// TIA Portal project "Poao_V21" (V21)

(* hardware
DEVICE "S7-1200 station_1"  S7-1200 Station
   slot 0: "Rack_0"  S7-1200 Rack  Rack  V1.0
   slot 1: "PLC_2"  CPU 1214C DC/DC/DC  6ES7 214-1AG40-0XB0  V4.4
DEVICE "PC station"  SIMATIC PC station
   slot 0: "PC station"  Rail  SIMATIC PC-Station  V1.0
      slot 125: "Stationmanager"  Station_Manager  V6.0.4
   slot 1: "IE general_1"  IE General  IE_CP  V8.2.0
      slot 1: "PROFINET interface"  IEGeneral.Interface.8.2.0
   slot 3: "HMI_RT_1"  WinCC RT Advanced  6AV2 104-0xxxx-xxxx  17.0.0.0
      slot 33792: "主机接口"  Host interface
*)

// ===== PLC "PLC_2"  CPU 1214C DC/DC/DC =====

VAR_GLOBAL   // PLC tag table "默认变量表"
   "1层外呼上行指示灯" AT %M24.0 : Bool;
   "2层外呼上行指示灯" AT %M24.1 : Bool;
   "3层外呼上行指示灯" AT %M24.2 : Bool;
   "4层外呼上行指示灯" AT %M24.3 : Bool;
   "5层外呼上行指示灯" AT %M24.4 : Bool;
   "2层外呼下行指示灯" AT %M24.5 : Bool;
   "3层外呼下行指示灯" AT %M24.6 : Bool;
   "4层外呼下行指示灯" AT %M24.7 : Bool;
   "6层外呼下行指示灯" AT %M25.1 : Bool;
   "1号梯1层内呼指示灯" AT %M25.2 : Bool;
   "1号梯2层内呼指示灯" AT %M25.3 : Bool;
   "1号梯3层内呼指示灯" AT %M25.4 : Bool;
   "1号梯4层内呼指示灯" AT %M25.5 : Bool;
   "1号梯5层内呼指示灯" AT %M25.6 : Bool;
   "1号梯6层内呼指示灯" AT %M25.7 : Bool;
   "1号梯七段数码管a" AT %M26.2 : Bool;
   "1号梯七段数码管b" AT %M26.3 : Bool;
   "1号梯七段数码管c" AT %M26.4 : Bool;
   "1号梯七段数码管d" AT %M26.5 : Bool;
   "1号梯七段数码管e" AT %M26.6 : Bool;
   "1号梯七段数码管f" AT %M26.7 : Bool;
   "1号梯七段数码管g" AT %M33.7 : Bool;
   "1号梯上行指示" AT %M23.4 : Bool;
   "1号梯下行指示" AT %M2.5 : Bool;
   "1号梯电机启动信号" AT %M2.6 : Bool;
   "1号梯故障指示" AT %M23.5 : Bool;
   "1号梯照明指示" AT %M23.6 : Bool;
   "1号梯风扇指示" AT %M23.7 : Bool;
   "1号梯高速运行" AT %M2.7 : Bool;
   "1号梯低速运行" AT %M405.7 : Bool;
   "1号梯1级制动接触器" AT %M5.5 : Bool;
   "1号梯2级制动接触器" AT %M5.6 : Bool;
   "1号梯3级制动接触器" AT %M10.7 : Bool;
   "1号梯满载指示" AT %M21.4 : Bool;
   "1号梯1层内选按钮" AT %M21.5 : Bool;
   "1号梯2层内选按钮" AT %M21.6 : Bool;
   "1号梯3层内选按钮" AT %M22.7 : Bool;
   "1号梯4层内选按钮" AT %M20.0 : Bool;
   "1号梯5层内选按钮" AT %M20.1 : Bool;
   "1号梯6层内选按钮" AT %M20.2 : Bool;
   "1层上行按钮" AT %M20.3 : Bool;
   "2层上行按钮" AT %M20.4 : Bool;
   "3层上行按钮" AT %M20.5 : Bool;
   "4层上行按钮" AT %M20.6 : Bool;
   "5层上行按钮" AT %M21.7 : Bool;
   "2层下行按钮" AT %M19.0 : Bool;
   "3层下行按钮" AT %M19.1 : Bool;
   "4层下行按钮" AT %M19.2 : Bool;
   "5层下行按钮" AT %M19.3 : Bool;
   "6层下行按钮" AT %M19.4 : Bool;
   "1号梯轿内开门按钮" AT %M19.5 : Bool;
   "1号梯轿内关门按钮" AT %M19.6 : Bool;
   "1号梯红外光幕信号" AT %M20.7 : Bool;
   "1号梯超重信号" AT %M16.0 : Bool;
   "1号梯检修开关" AT %M16.1 : Bool;
   "1号梯轿厢门锁信号" AT %M409.4 : Bool;
   "1号梯1层门锁信号" AT %M16.3 : Bool;
   "1号梯2层门锁信号" AT %M16.4 : Bool;
   "1号梯3层门锁信号" AT %M16.5 : Bool;
   "1号梯4层门锁信号" AT %M16.6 : Bool;
   "1号梯5层门锁信号" AT %M16.7 : Bool;
   "1号梯6层门锁信号" AT %M17.0 : Bool;
   "1号梯开门到位" AT %M17.1 : Bool;
   "1号梯关门到位" AT %M17.2 : Bool;
   "1号梯上平层信号" AT %M17.3 : Bool;
   "1号梯下平层信号" AT %M17.4 : Bool;
   "1号梯上端站第1限位" AT %M17.5 : Bool;
   "1号梯上端站第2限位" AT %M17.6 : Bool;
   "1号梯下端站第1限位" AT %M17.7 : Bool;
   "1号梯下端站第2限位" AT %M18.0 : Bool;
   "自动运行信号" AT %M10.1 : Bool;
   "沿0" AT %M10.2 : Bool;
   "沿4" AT %M10.3 : Bool;
   "沿5" AT %M10.4 : Bool;
   "沿6" AT %M10.5 : Bool;
   "沿7" AT %M10.6 : Bool;
   "沿9" AT %M19.7 : Bool;
   "沿10" AT %M500.0 : Bool;
   "沿500" AT %M500.1 : Bool;
   "沿501" AT %M500.2 : Bool;
   "沿13" AT %M500.3 : Bool;
   "沿14" AT %M500.4 : Bool;
   "沿15" AT %M500.5 : Bool;
   "沿16" AT %M500.6 : Bool;
   "沿17" AT %M500.7 : Bool;
   "沿18" AT %M501.0 : Bool;
   "沿19" AT %M501.1 : Bool;
   "沿20" AT %M501.2 : Bool;
   "1号梯低速转高速" AT %M501.3 : Bool;
   "1号梯制动使能" AT %M501.4 : Bool;
   "1号梯制动完成" AT %M501.5 : Bool;
   "沿27" AT %M503.1 : Bool;
   "沿29" AT %M503.3 : Bool;
   "沿30" AT %M13.4 : Bool;
   "沿31" AT %M13.5 : Bool;
   "沿32" AT %M13.6 : Bool;
   "沿33" AT %M13.7 : Bool;
   "沿34" AT %M14.0 : Bool;
   "沿35" AT %M14.1 : Bool;
   "1号梯准备就绪标志位" AT %M14.2 : Bool;
   "沿37" AT %M14.3 : Bool;
   "沿38" AT %M14.4 : Bool;
   "沿39" AT %M14.5 : Bool;
   "沿40" AT %M14.6 : Bool;
   "沿41" AT %M14.7 : Bool;
   "沿50" AT %M15.0 : Bool;
   "沿51" AT %M15.1 : Bool;
   "沿52" AT %M15.2 : Bool;
   "沿53" AT %M15.3 : Bool;
   "上沿1" AT %M16.2 : Bool;
   "上沿2" AT %M18.1 : Bool;
   "上沿3" AT %M18.2 : Bool;
   "上沿4" AT %M18.3 : Bool;
   "上沿5" AT %M18.4 : Bool;
   "上沿6" AT %M18.5 : Bool;
   "下沿1" AT %M18.6 : Bool;
   "下沿2" AT %M18.7 : Bool;
   "下沿3" AT %M21.0 : Bool;
   "下沿4" AT %M21.1 : Bool;
   "下沿5" AT %M21.2 : Bool;
   "下沿6" AT %M21.3 : Bool;
   "内沿1" AT %M22.0 : Bool;
   "内沿2" AT %M22.1 : Bool;
   "内沿3" AT %M22.2 : Bool;
   "内沿4" AT %M22.3 : Bool;
   "内沿5" AT %M22.4 : Bool;
   "内沿6" AT %M22.5 : Bool;
   "1号梯高速转低速" AT %M202.7 : Bool;
   "6层上行按钮" AT %M22.6 : Bool;
   "7层上行按钮" AT %M60.6 : Bool;
   "7层下行按钮" AT %M60.4 : Bool;
   "1号梯7层内呼指示灯" AT %M60.7 : Bool;
   "1号梯7层内选按钮" AT %M60.2 : Bool;
   "7层外呼下行指示灯" AT %M60.1 : Bool;
   "1号梯7层门锁信号" AT %M60.0 : Bool;
   "8层上行按钮" AT %M61.6 : Bool;
   "8层下行按钮" AT %M61.4 : Bool;
   "1号梯8层内呼指示灯" AT %M61.7 : Bool;
   "1号梯8层内选按钮" AT %M61.2 : Bool;
   "8层外呼下行指示灯" AT %M61.1 : Bool;
   "1号梯8层门锁信号" AT %M61.0 : Bool;
   "9层上行按钮" AT %M62.6 : Bool;
   "9层下行按钮" AT %M62.4 : Bool;
   "1号梯9层内呼指示灯" AT %M62.7 : Bool;
   "1号梯9层内选按钮" AT %M62.2 : Bool;
   "9层外呼下行指示灯" AT %M62.1 : Bool;
   "1号梯9层门锁信号" AT %M62.0 : Bool;
   "10层下行按钮" AT %M63.4 : Bool;
   "1号梯10层内呼指示灯" AT %M63.7 : Bool;
   "1号梯10层内选按钮" AT %M63.2 : Bool;
   "10层外呼下行指示灯" AT %M63.1 : Bool;
   "1号梯10层门锁信号" AT %M63.0 : Bool;
   "沿1" AT %M23.1 : Bool;
   "沿3" AT %M23.2 : Bool;
   "1号梯向上回一楼信号" AT %M3.1 : Bool;
   "1号梯向下回一楼信号" AT %M3.2 : Bool;
   "5层外呼下行指示灯" AT %M25.0 : Bool;
   "7层外呼上行指示灯" AT %M34.4 : Bool;
   "6层外呼上行指示灯" AT %M34.6 : Bool;
   "10层外呼上行指示灯" AT %M35.1 : Bool;
   "8层外呼上行指示灯" AT %M34.5 : Bool;
   "9层外呼上行指示灯" AT %M34.7 : Bool;
   "1号梯七段数码管h" AT %M33.0 : Bool;
   "1号梯七段数码管n" AT %M23.0 : Bool;
   "1号梯七段数码管m" AT %M33.5 : Bool;
   "1号梯七段数码管i" AT %M33.1 : Bool;
   "1号梯七段数码管l" AT %M33.4 : Bool;
   "1号梯七段数码管j" AT %M33.2 : Bool;
   "1号梯七段数码管k" AT %M33.3 : Bool;
   "沿100" AT %M33.6 : Bool;
   "沿101" AT %M34.0 : Bool;
   "沿102" AT %M34.1 : Bool;
   "沿103" AT %M34.2 : Bool;
   "沿104" AT %M34.3 : Bool;
   "沿105" AT %M35.0 : Bool;
   "沿106" AT %M35.2 : Bool;
   "沿107" AT %M35.3 : Bool;
   "1号梯6层上呼" AT %M35.4 : Bool;
   "1号梯7层上呼" AT %M35.5 : Bool;
   "1号梯8层上呼" AT %M35.6 : Bool;
   "1号梯9层上呼" AT %M35.7 : Bool;
   "1号梯7层下呼" AT %M36.0 : Bool;
   "1号梯8层下呼" AT %M36.1 : Bool;
   "1号梯9层下呼" AT %M36.2 : Bool;
   "1号梯10层下呼" AT %M36.3 : Bool;
   "上沿7" AT %M23.3 : Bool;
   "上沿8" AT %M26.0 : Bool;
   "上沿9" AT %M26.1 : Bool;
   "下沿7" AT %M27.0 : Bool;
   "下沿8" AT %M27.1 : Bool;
   "下沿9" AT %M27.2 : Bool;
   "下沿10" AT %M27.3 : Bool;
   "内沿7" AT %M27.4 : Bool;
   "内沿8" AT %M27.5 : Bool;
   "内沿9" AT %M27.6 : Bool;
   "内沿10" AT %M27.7 : Bool;
   "1号梯1层灭灯" AT %M28.0 : Bool;
   "1号梯1层指示灯控制" AT %MW700 : Int;
   "1号梯2层指示灯控制" AT %MW702 : Int;
   "1号梯3层指示灯控制" AT %MW704 : Int;
   "1号梯4层指示灯控制" AT %MW706 : Int;
   "1号梯5层指示灯控制" AT %MW708 : Int;
   "1号梯6层指示灯控制" AT %MW710 : Int;
   "1号梯7层指示灯控制" AT %MW7501 : Int;
   "1号梯8层指示灯控制" AT %MW714 : Int;
   "1号梯9层指示灯控制" AT %MW716 : Int;
   "1号梯10层指示灯控制" AT %MW718 : Int;
   "1号梯2层灭灯" AT %M800.0 : Bool;
   "1号梯3层灭灯" AT %M802.0 : Bool;
   "1号梯4层灭灯" AT %M802.1 : Bool;
   "1号梯5层灭灯" AT %M802.2 : Bool;
   "1号梯6层灭灯" AT %M802.3 : Bool;
   "1号梯7层灭灯" AT %M802.4 : Bool;
   "1号梯8层灭灯" AT %M802.5 : Bool;
   "1号梯9层灭灯" AT %M802.6 : Bool;
   "1号梯10层灭灯" AT %M802.7 : Bool;
   "1号梯超重信号沿" AT %M803.0 : Bool;
   "1号梯故障指示灯闪烁中间变量" AT %M1.0 : Bool;
   "1号梯标量化" AT %MD5010 : Real;
   "1号梯故障开关沿" AT %M200.0 : Bool;
   "1号梯检修开关沿" AT %M200.1 : Bool;
   "1号梯检修开关沿2" AT %M200.2 : Bool;
END_VAR

VAR_GLOBAL   // PLC tag table "电梯变量表"
   "1号梯当前楼层数" AT %MW2000 : Int;
   "1号梯上行命令" AT %M2.0 : Bool;
   "1号梯下行命令" AT %M2.1 : Bool;
   "1号梯电梯静止" AT %M3.0 : Bool;
   "1号梯平层信号" AT %M3.3 : Bool;
   "1号梯门锁确认信号" AT %M3.4 : Bool;
   "1号梯电梯停稳信号" AT %M3.5 : Bool;
   "1号梯登记1层" AT %M4.0 : Bool;
   "1号梯登记2层" AT %M4.1 : Bool;
   "1号梯登记3层" AT %M4.2 : Bool;
   "1号梯登记4层" AT %M4.3 : Bool;
   "1号梯登记5层" AT %M4.4 : Bool;
   "1号梯登记6层" AT %M4.5 : Bool;
   "1号梯电梯休眠信号" AT %M3.6 : Bool;
   "1号梯准备就绪信号" AT %M4.6 : Bool;
   "1号梯开门锁上下行" AT %M4.7 : Bool;
   "1号梯本层召唤开门信号" AT %M5.0 : Bool;
   "1号梯上行呼叫标志位" AT %M5.1 : Bool;
   "1号梯下行呼叫标志位" AT %M5.2 : Bool;
   "1号梯上行接触器" AT %M5.3 : Bool;
   "1号梯下行接触器" AT %M5.4 : Bool;
   "1号梯开门继电器" AT %M5.7 : Bool;
   "1号梯关门继电器" AT %M6.0 : Bool;
   "1号梯1层上呼" AT %M6.1 : Bool;
   "1号梯2层上呼" AT %M6.2 : Bool;
   "1号梯3层上呼" AT %M6.3 : Bool;
   "1号梯4层上呼" AT %M6.4 : Bool;
   "1号梯5层上呼" AT %M6.5 : Bool;
   "1号梯2层下呼" AT %M6.6 : Bool;
   "1号梯3层下呼" AT %M6.7 : Bool;
   "1号梯4层下呼" AT %M7.0 : Bool;
   "1号梯5层下呼" AT %M7.1 : Bool;
   "1号梯6层下呼" AT %M7.2 : Bool;
   "1号梯休眠信号" AT %M7.7 : Bool;
   "1号梯向下初始化信号" AT %M8.2 : Bool;
   "2号梯电梯当前载重" AT %MW800 : Int;
   "1号梯向上初始化信号" AT %M255.2 : Bool;
   "1号梯电梯当前载重" AT %MW720 : Int;
   "3号梯电梯当前载重" AT %MW850 : Int;
   "1号梯登记7层" AT %M7.3 : Bool;
   "1号梯登记8层" AT %M7.4 : Bool;
   "1号梯登记9层" AT %M7.5 : Bool;
   "1号梯登记10层" AT %M7.6 : Bool;
END_VAR

VAR_GLOBAL   // PLC tag table "2号梯变量表"
   "2号梯高速转低速" AT %M0.3 : Bool;
   "2号梯准备就绪标志位" AT %M3.7 : Bool;
   "2号梯制动完成" AT %M505.0 : Bool;
   "2号梯制动使能" AT %M505.1 : Bool;
   "2号梯低速转高速" AT %M505.2 : Bool;
   "2号梯下端站第2限位" AT %M705.5 : Bool;
   "2号梯下端站第1限位" AT %M507.6 : Bool;
   "2号梯上端站第2限位" AT %M507.7 : Bool;
   "2号梯上端站第1限位" AT %M8.0 : Bool;
   "2号梯下平层信号" AT %M8.1 : Bool;
   "2号梯上平层信号" AT %M508.2 : Bool;
   "2号梯关门到位" AT %M8.3 : Bool;
   "2号梯开门到位" AT %M8.4 : Bool;
   "2号梯6层门锁信号" AT %M8.5 : Bool;
   "2号梯5层门锁信号" AT %M8.6 : Bool;
   "2号梯4层门锁信号" AT %M8.7 : Bool;
   "2号梯3层门锁信号" AT %M9.0 : Bool;
   "2号梯2层门锁信号" AT %M9.1 : Bool;
   "2号梯1层门锁信号" AT %M9.2 : Bool;
   "2号梯轿厢门锁信号" AT %M9.3 : Bool;
   "2号梯检修开关" AT %M9.4 : Bool;
   "2号梯超重信号" AT %M9.5 : Bool;
   "2号梯红外光幕信号" AT %M9.6 : Bool;
   "2号梯轿内关门按钮" AT %M9.7 : Bool;
   "2号梯轿内开门按钮" AT %M10.0 : Bool;
   "2号梯6层内选按钮" AT %M11.3 : Bool;
   "2号梯5层内选按钮" AT %M11.4 : Bool;
   "2号梯4层内选按钮" AT %M11.5 : Bool;
   "2号梯3层内选按钮" AT %M11.6 : Bool;
   "2号梯2层内选按钮" AT %M11.7 : Bool;
   "2号梯1层内选按钮" AT %M12.0 : Bool;
   "2号梯满载指示" AT %M12.1 : Bool;
   "2号梯3级制动接触器" AT %M12.2 : Bool;
   "2号梯2级制动接触器" AT %M12.3 : Bool;
   "2号梯1级制动接触器" AT %M12.4 : Bool;
   "2号梯低速运行" AT %M12.5 : Bool;
   "2号梯高速运行" AT %M12.6 : Bool;
   "2号梯风扇指示" AT %M12.7 : Bool;
   "2号梯照明指示" AT %M13.0 : Bool;
   "2号梯故障指示" AT %M13.1 : Bool;
   "2号梯电机启动信号" AT %M13.2 : Bool;
   "2号梯下行指示" AT %M13.3 : Bool;
   "2号梯上行指示" AT %M900.4 : Bool;
   "2号梯七段数码管g" AT %M900.5 : Bool;
   "2号梯七段数码管f" AT %M900.6 : Bool;
   "2号梯七段数码管e" AT %M900.7 : Bool;
   "2号梯七段数码管d" AT %M901.0 : Bool;
   "2号梯七段数码管c" AT %M901.1 : Bool;
   "2号梯七段数码管b" AT %M901.2 : Bool;
   "2号梯七段数码管a" AT %M901.3 : Bool;
   "2号梯6层内呼指示灯" AT %M901.4 : Bool;
   "2号梯5层内呼指示灯" AT %M901.5 : Bool;
   "2号梯4层内呼指示灯" AT %M901.6 : Bool;
   "2号梯3层内呼指示灯" AT %M901.7 : Bool;
   "2号梯2层内呼指示灯" AT %M902.0 : Bool;
   "2号梯1层内呼指示灯" AT %M902.1 : Bool;
   "2号梯7层内呼指示灯" AT %M903.0 : Bool;
   "2号梯7层内选按钮" AT %M903.1 : Bool;
   "2号梯7层门锁信号" AT %M903.3 : Bool;
   "2号梯8层内呼指示灯" AT %M903.6 : Bool;
   "2号梯8层内选按钮" AT %M903.7 : Bool;
   "2号梯8层门锁信号" AT %M904.1 : Bool;
   "2号梯9层内呼指示灯" AT %M904.4 : Bool;
   "2号梯9层内选按钮" AT %M904.5 : Bool;
   "2号梯9层门锁信号" AT %M904.7 : Bool;
   "2号梯10层内呼指示灯" AT %M905.1 : Bool;
   "2号梯10层内选按钮" AT %M905.2 : Bool;
   "2号梯10层门锁信号" AT %M905.4 : Bool;
   "2号梯向上回一楼信号" AT %M905.7 : Bool;
   "2号梯向下回一楼信号" AT %M906.0 : Bool;
   "2号梯七段数码管h" AT %M43.0 : Bool;
   "2号梯七段数码管n" AT %M43.1 : Bool;
   "2号梯七段数码管m" AT %M43.5 : Bool;
   "2号梯七段数码管i" AT %M43.2 : Bool;
   "2号梯七段数码管l" AT %M43.4 : Bool;
   "2号梯七段数码管j" AT %M43.6 : Bool;
   "2号梯七段数码管k" AT %M43.3 : Bool;
   "2号梯上行接触器" AT %M43.7 : Bool;
   "2号梯下行接触器" AT %M44.0 : Bool;
   "2号梯开门锁上下行" AT %M44.1 : Bool;
   "2号梯开门继电器" AT %M44.2 : Bool;
   "2号梯关门继电器" AT %M44.3 : Bool;
   "2号梯准备就绪信号" AT %M44.4 : Bool;
   "2号梯当前楼层数" AT %MW2100 : Int;
   "2号梯上行命令" AT %M610.0 : Bool;
   "2号梯上行呼叫标志位" AT %M610.1 : Bool;
   "2号梯下行命令" AT %M610.2 : Bool;
   "2号梯1层上呼" AT %M610.3 : Bool;
   "2号梯2层上呼" AT %M610.4 : Bool;
   "2号梯3层上呼" AT %M610.5 : Bool;
   "2号梯4层上呼" AT %M610.6 : Bool;
   "2号梯5层上呼" AT %M610.7 : Bool;
   "2号梯6层上呼" AT %M36.4 : Bool;
   "2号梯7层上呼" AT %M36.5 : Bool;
   "2号梯8层上呼" AT %M36.6 : Bool;
   "2号梯9层上呼" AT %M36.7 : Bool;
   "2号梯下行呼叫标志位" AT %M37.0 : Bool;
   "2号梯2层下呼" AT %M37.1 : Bool;
   "2号梯3层下呼" AT %M37.2 : Bool;
   "2号梯4层下呼" AT %M37.3 : Bool;
   "2号梯5层下呼" AT %M37.4 : Bool;
   "2号梯6层下呼" AT %M37.5 : Bool;
   "2号梯7层下呼" AT %M37.6 : Bool;
   "2号梯8层下呼" AT %M37.7 : Bool;
   "2号梯9层下呼" AT %M38.0 : Bool;
   "2号梯10层下呼" AT %M38.1 : Bool;
   "2号梯向下初始化信号" AT %M38.2 : Bool;
   "2号梯向上初始化信号" AT %M38.3 : Bool;
   "2号梯休眠信号" AT %M38.4 : Bool;
   "2号梯登记1层" AT %M38.5 : Bool;
   "2号梯登记2层" AT %M38.6 : Bool;
   "2号梯登记3层" AT %M38.7 : Bool;
   "2号梯登记4层" AT %M39.0 : Bool;
   "2号梯登记5层" AT %M39.1 : Bool;
   "2号梯登记6层" AT %M39.2 : Bool;
   "2号梯登记7层" AT %M39.3 : Bool;
   "2号梯登记8层" AT %M39.4 : Bool;
   "2号梯登记9层" AT %M39.5 : Bool;
   "2号梯登记10层" AT %M39.6 : Bool;
   "2号梯本层召唤开门信号" AT %M39.7 : Bool;
   "2号梯门锁确认信号" AT %M40.0 : Bool;
   "2号梯平层信号" AT %M40.1 : Bool;
   "2号梯电梯停稳信号" AT %M40.2 : Bool;
   "沿200" AT %M40.3 : Bool;
   "沿201" AT %M40.4 : Bool;
   "沿202" AT %M40.5 : Bool;
   "沿203" AT %M40.6 : Bool;
   "沿204" AT %M40.7 : Bool;
   "沿205" AT %M41.0 : Bool;
   "沿206" AT %M41.1 : Bool;
   "沿207" AT %M41.2 : Bool;
   "沿208" AT %M41.3 : Bool;
   "沿209" AT %M41.4 : Bool;
   "沿210" AT %M41.5 : Bool;
   "沿211" AT %M41.6 : Bool;
   "沿212" AT %M41.7 : Bool;
   "沿213" AT %M44.5 : Bool;
   "沿2901" AT %M44.6 : Bool;
   "沿2902" AT %M44.7 : Bool;
   "沿216" AT %M45.0 : Bool;
   "沿217" AT %M45.1 : Bool;
   "沿218" AT %M45.2 : Bool;
   "沿219" AT %M45.3 : Bool;
   "沿220" AT %M45.4 : Bool;
   "沿221" AT %M45.5 : Bool;
   "沿222" AT %M45.6 : Bool;
   "沿223" AT %M45.7 : Bool;
   "沿224" AT %M46.0 : Bool;
   "沿225" AT %M46.1 : Bool;
   "沿226" AT %M46.2 : Bool;
   "沿227" AT %M46.3 : Bool;
   "沿228" AT %M50.3 : Bool;
   "沿229" AT %M50.4 : Bool;
   "沿230" AT %M50.5 : Bool;
   "沿231" AT %M50.6 : Bool;
   "沿232" AT %M50.7 : Bool;
   "沿2903" AT %M51.0 : Bool;
   "沿2904" AT %M51.1 : Bool;
   "沿2905" AT %M51.2 : Bool;
   "沿236" AT %M51.3 : Bool;
   "沿237" AT %M51.4 : Bool;
   "沿238" AT %M51.5 : Bool;
   "沿239" AT %M51.6 : Bool;
   "2号梯2层灭灯" AT %M58.4 : Bool;
   "2号梯3层灭灯" AT %M58.5 : Bool;
   "2号梯4层灭灯" AT %M58.6 : Bool;
   "2号梯1层灭灯" AT %M58.7 : Bool;
   "2号梯5层灭灯" AT %M59.0 : Bool;
   "2号梯6层灭灯" AT %M59.1 : Bool;
   "2号梯7层灭灯" AT %M59.2 : Bool;
   "2号梯8层灭灯" AT %M59.3 : Bool;
   "2号梯9层灭灯" AT %M59.4 : Bool;
   "2号梯10层灭灯" AT %M59.5 : Bool;
   "2号梯1层指示灯控制" AT %MW2200 : Int;
   "2号梯2层指示灯控制" AT %MW2202 : Int;
   "2号梯3层指示灯控制" AT %MW2204 : Int;
   "2号梯4层指示灯控制" AT %MW2206 : Int;
   "2号梯5层指示灯控制" AT %MW2208 : Int;
   "2号梯6层指示灯控制" AT %MW2210 : Int;
   "2号梯7层指示灯控制" AT %MW2212 : Int;
   "2号梯8层指示灯控制" AT %MW2201 : Int;
   "2号梯9层指示灯控制" AT %MW2216 : Int;
   "2号梯10层指示灯控制" AT %MW2218 : Int;
   "内沿20" AT %M90.0 : Bool;
   "内沿21" AT %M90.1 : Bool;
   "内沿22" AT %M90.2 : Bool;
   "内沿23" AT %M90.3 : Bool;
   "内沿24" AT %M90.4 : Bool;
   "内沿25" AT %M90.5 : Bool;
   "内沿26" AT %M90.6 : Bool;
   "内沿27" AT %M90.7 : Bool;
   "内沿28" AT %M91.0 : Bool;
   "内沿29" AT %M91.1 : Bool;
   "2号梯超重信号沿" AT %M91.2 : Bool;
   "2号梯故障指示灯闪烁中间变量" AT %M91.3 : Bool;
   "2号梯标量化" AT %MD122 : Real;
   "2号梯故障开关沿" AT %M201.0 : Bool;
   "2号梯检修开关沿" AT %M201.1 : Bool;
   "2号梯检修开关沿2" AT %M201.2 : Bool;
END_VAR

VAR_GLOBAL   // PLC tag table "3号梯变量表"
   "3号梯向下回一楼信号" AT %M400.2 : Bool;
   "3号梯向上回一楼信号" AT %M400.3 : Bool;
   "3号梯10层门锁信号" AT %M400.4 : Bool;
   "3号梯10层内选按钮" AT %M400.5 : Bool;
   "3号梯10层内呼指示灯" AT %M400.6 : Bool;
   "3号梯9层门锁信号" AT %M400.7 : Bool;
   "3号梯9层内选按钮" AT %M401.0 : Bool;
   "3号梯9层内呼指示灯" AT %M401.1 : Bool;
   "3号梯8层门锁信号" AT %M401.2 : Bool;
   "3号梯8层内选按钮" AT %M401.3 : Bool;
   "3号梯8层内呼指示灯" AT %M401.4 : Bool;
   "3号梯7层门锁信号" AT %M401.5 : Bool;
   "3号梯7层内选按钮" AT %M401.6 : Bool;
   "3号梯7层内呼指示灯" AT %M401.7 : Bool;
   "3号梯1层内呼指示灯" AT %M402.0 : Bool;
   "3号梯2层内呼指示灯" AT %M402.1 : Bool;
   "3号梯3层内呼指示灯" AT %M402.2 : Bool;
   "3号梯4层内呼指示灯" AT %M402.3 : Bool;
   "3号梯5层内呼指示灯" AT %M402.4 : Bool;
   "3号梯6层内呼指示灯" AT %M402.5 : Bool;
   "3号梯七段数码管a" AT %M402.6 : Bool;
   "3号梯七段数码管b" AT %M402.7 : Bool;
   "3号梯七段数码管c" AT %M403.0 : Bool;
   "3号梯七段数码管d" AT %M403.1 : Bool;
   "3号梯七段数码管e" AT %M403.2 : Bool;
   "3号梯七段数码管f" AT %M403.3 : Bool;
   "3号梯七段数码管g" AT %M403.4 : Bool;
   "3号梯上行指示" AT %M403.5 : Bool;
   "3号梯下行指示" AT %M403.6 : Bool;
   "3号梯电机启动信号" AT %M403.7 : Bool;
   "3号梯故障指示" AT %M88.0 : Bool;
   "3号梯照明指示" AT %M28.1 : Bool;
   "3号梯风扇指示" AT %M28.2 : Bool;
   "3号梯高速运行" AT %M28.3 : Bool;
   "3号梯低速运行" AT %M28.4 : Bool;
   "3号梯1级制动接触器" AT %M28.5 : Bool;
   "3号梯2级制动接触器" AT %M28.6 : Bool;
   "3号梯3级制动接触器" AT %M28.7 : Bool;
   "3号梯满载指示" AT %M29.0 : Bool;
   "3号梯1层内选按钮" AT %M29.1 : Bool;
   "3号梯2层内选按钮" AT %M29.2 : Bool;
   "3号梯3层内选按钮" AT %M29.3 : Bool;
   "3号梯4层内选按钮" AT %M29.4 : Bool;
   "3号梯5层内选按钮" AT %M29.5 : Bool;
   "3号梯6层内选按钮" AT %M29.6 : Bool;
   "3号梯轿内开门按钮" AT %M29.7 : Bool;
   "3号梯轿内关门按钮" AT %M30.0 : Bool;
   "3号梯红外光幕信号" AT %M30.1 : Bool;
   "3号梯超重信号" AT %M30.2 : Bool;
   "3号梯检修开关" AT %M30.3 : Bool;
   "3号梯轿厢门锁信号" AT %M30.4 : Bool;
   "3号梯1层门锁信号" AT %M30.5 : Bool;
   "3号梯2层门锁信号" AT %M30.6 : Bool;
   "3号梯3层门锁信号" AT %M30.7 : Bool;
   "3号梯4层门锁信号" AT %M31.0 : Bool;
   "3号梯5层门锁信号" AT %M31.1 : Bool;
   "3号梯6层门锁信号" AT %M31.2 : Bool;
   "3号梯开门到位" AT %M31.3 : Bool;
   "3号梯关门到位" AT %M31.4 : Bool;
   "3号梯上平层信号" AT %M31.5 : Bool;
   "3号梯下平层信号" AT %M31.6 : Bool;
   "3号梯上端站第1限位" AT %M31.7 : Bool;
   "3号梯上端站第2限位" AT %M32.0 : Bool;
   "3号梯下端站第1限位" AT %M32.1 : Bool;
   "3号梯下端站第2限位" AT %M32.2 : Bool;
   "3号梯低速转高速" AT %M32.3 : Bool;
   "3号梯制动使能" AT %M32.4 : Bool;
   "3号梯制动完成" AT %M32.5 : Bool;
   "3号梯准备就绪标志位" AT %M32.6 : Bool;
   "3号梯高速转低速" AT %M32.7 : Bool;
   "3号梯七段数码管h" AT %M53.0 : Bool;
   "3号梯七段数码管n" AT %M53.6 : Bool;
   "3号梯七段数码管m" AT %M53.5 : Bool;
   "3号梯七段数码管i" AT %M53.1 : Bool;
   "3号梯七段数码管l" AT %M53.4 : Bool;
   "3号梯七段数码管j" AT %M53.2 : Bool;
   "3号梯七段数码管k" AT %M53.3 : Bool;
   "3号梯上行接触器" AT %M53.7 : Bool;
   "3号梯下行接触器" AT %M54.0 : Bool;
   "3号梯开门锁上下行" AT %M54.1 : Bool;
   "3号梯开门继电器" AT %M54.2 : Bool;
   "3号梯关门继电器" AT %M54.3 : Bool;
   "3号梯准备就绪信号" AT %M54.4 : Bool;
   "3号梯当前楼层数" AT %MW2300 : Int;
   "3号梯上行命令" AT %M42.0 : Bool;
   "3号梯上行呼叫标志位" AT %M42.1 : Bool;
   "3号梯下行命令" AT %M42.2 : Bool;
   "3号梯1层上呼" AT %M42.3 : Bool;
   "3号梯2层上呼" AT %M42.4 : Bool;
   "3号梯3层上呼" AT %M42.5 : Bool;
   "3号梯4层上呼" AT %M42.6 : Bool;
   "3号梯5层上呼" AT %M42.7 : Bool;
   "3号梯6层上呼" AT %M46.4 : Bool;
   "3号梯7层上呼" AT %M46.5 : Bool;
   "3号梯8层上呼" AT %M46.6 : Bool;
   "3号梯9层上呼" AT %M46.7 : Bool;
   "3号梯下行呼叫标志位" AT %M47.0 : Bool;
   "3号梯2层下呼" AT %M47.1 : Bool;
   "3号梯3层下呼" AT %M47.2 : Bool;
   "3号梯4层下呼" AT %M47.3 : Bool;
   "3号梯5层下呼" AT %M47.4 : Bool;
   "3号梯6层下呼" AT %M47.5 : Bool;
   "3号梯7层下呼" AT %M47.6 : Bool;
   "3号梯8层下呼" AT %M47.7 : Bool;
   "3号梯9层下呼" AT %M48.0 : Bool;
   "3号梯10层下呼" AT %M48.1 : Bool;
   "3号梯向下初始化信号" AT %M48.2 : Bool;
   "3号梯向上初始化信号" AT %M48.3 : Bool;
   "3号梯休眠信号" AT %M48.4 : Bool;
   "3号梯登记1层" AT %M48.5 : Bool;
   "3号梯登记2层" AT %M48.6 : Bool;
   "3号梯登记3层" AT %M48.7 : Bool;
   "3号梯登记4层" AT %M49.0 : Bool;
   "3号梯登记5层" AT %M49.1 : Bool;
   "3号梯登记6层" AT %M49.2 : Bool;
   "3号梯登记7层" AT %M49.3 : Bool;
   "3号梯登记8层" AT %M49.4 : Bool;
   "3号梯登记9层" AT %M49.5 : Bool;
   "3号梯登记10层" AT %M49.6 : Bool;
   "3号梯本层召唤开门信号" AT %M49.7 : Bool;
   "3号梯门锁确认信号" AT %M50.0 : Bool;
   "3号梯平层信号" AT %M50.1 : Bool;
   "3号梯电梯停稳信号" AT %M50.2 : Bool;
   "沿300" AT %M51.7 : Bool;
   "沿301" AT %M52.0 : Bool;
   "沿302" AT %M52.1 : Bool;
   "沿303" AT %M52.2 : Bool;
   "沿304" AT %M52.3 : Bool;
   "沿305" AT %M52.4 : Bool;
   "沿306" AT %M52.5 : Bool;
   "沿307" AT %M52.6 : Bool;
   "沿308" AT %M52.7 : Bool;
   "沿309" AT %M54.5 : Bool;
   "沿310" AT %M54.6 : Bool;
   "沿311" AT %M54.7 : Bool;
   "沿312" AT %M55.0 : Bool;
   "沿313" AT %M55.1 : Bool;
   "沿314" AT %M55.2 : Bool;
   "沿315" AT %M55.3 : Bool;
   "沿316" AT %M55.4 : Bool;
   "沿317" AT %M55.5 : Bool;
   "沿318" AT %M55.6 : Bool;
   "沿319" AT %M55.7 : Bool;
   "沿320" AT %M56.0 : Bool;
   "沿321" AT %M56.1 : Bool;
   "沿322" AT %M56.2 : Bool;
   "沿323" AT %M56.3 : Bool;
   "沿3400" AT %M56.4 : Bool;
   "沿3401" AT %M56.5 : Bool;
   "沿3402" AT %M56.6 : Bool;
   "沿3403" AT %M56.7 : Bool;
   "沿328" AT %M57.0 : Bool;
   "沿329" AT %M57.1 : Bool;
   "沿330" AT %M57.2 : Bool;
   "沿331" AT %M57.3 : Bool;
   "沿332" AT %M57.4 : Bool;
   "沿333" AT %M57.5 : Bool;
   "沿334" AT %M57.6 : Bool;
   "沿335" AT %M57.7 : Bool;
   "沿336" AT %M58.0 : Bool;
   "沿337" AT %M58.1 : Bool;
   "沿338" AT %M58.2 : Bool;
   "沿339" AT %M58.3 : Bool;
   "3号梯1层灭灯" AT %M59.6 : Bool;
   "3号梯2层灭灯" AT %M59.7 : Bool;
   "3号梯3层灭灯" AT %M60.3 : Bool;
   "3号梯4层灭灯" AT %M60.5 : Bool;
   "3号梯5层灭灯" AT %M61.3 : Bool;
   "3号梯6层灭灯" AT %M61.5 : Bool;
   "3号梯7层灭灯" AT %M62.3 : Bool;
   "3号梯8层灭灯" AT %M62.5 : Bool;
   "3号梯9层灭灯" AT %M63.3 : Bool;
   "3号梯10层灭灯" AT %M63.5 : Bool;
   "3号梯1层指示灯控制" AT %MW1000 : Int;
   "3号梯2层指示灯控制" AT %MW1002 : Int;
   "3号梯3层指示灯控制" AT %MW1004 : Int;
   "3号梯4层指示灯控制" AT %MW1006 : Int;
   "3号梯5层指示灯控制" AT %MW1008 : Int;
   "3号梯6层指示灯控制" AT %MW1010 : Int;
   "3号梯7层指示灯控制" AT %MW1012 : Int;
   "3号梯8层指示灯控制" AT %MW1014 : Int;
   "3号梯9层指示灯控制" AT %MW1016 : Int;
   "3号梯10层指示灯控制" AT %MW1018 : Int;
   "内沿30" AT %M100.0 : Bool;
   "内沿31" AT %M100.1 : Bool;
   "内沿32" AT %M100.2 : Bool;
   "内沿33" AT %M100.3 : Bool;
   "内沿34" AT %M100.4 : Bool;
   "内沿35" AT %M100.5 : Bool;
   "内沿36" AT %M100.6 : Bool;
   "内沿37" AT %M100.7 : Bool;
   "内沿38" AT %M101.0 : Bool;
   "内沿39" AT %M101.1 : Bool;
   "3号梯超重信号沿" AT %M101.2 : Bool;
   "3号梯故障指示灯闪烁中间变量" AT %M101.3 : Bool;
   "3号梯标量化" AT %MD121 : Real;
   "3号梯故障开关沿" AT %M202.0 : Bool;
   "3号梯检修开关沿" AT %M202.1 : Bool;
   "3号梯检修开关沿2" AT %M202.2 : Bool;
END_VAR

VAR_GLOBAL   // PLC tag table "变量表_1"
   "消防信号" AT %M1200.0 : Bool;
   "消防后关门" AT %M1200.1 : Bool;
   "消防信号下降沿" AT %M1200.2 : Bool;
   "1号梯消防信号的平层信号" AT %M1200.3 : Bool;
   "2号梯消防信号的平层信号" AT %M1200.4 : Bool;
   "3号梯消防信号的平层信号" AT %M1200.5 : Bool;
   "1号梯消防信号后初始化后" AT %M1200.6 : Bool;
   "2号梯消防信号后初始化后" AT %M1200.7 : Bool;
   "3号梯消防信号后初始化后" AT %M1201.0 : Bool;
   "1号梯独立运行模式" AT %M1201.1 : Bool;
   "2号梯独立运行模式" AT %M1201.2 : Bool;
   "3号梯独立运行模式" AT %M1201.3 : Bool;
   "第二次自动运行信号" AT %M1201.4 : Bool;
   "向上初始化使能" AT %M1201.5 : Bool;
END_VAR

DATA_BLOCK "input"   // DB10
{ S7_Optimized_Access := 'FALSE' }
VERSION : 0.1
   VAR
      "1层上行呼梯按钮" : Bool;
      "2层上行呼梯按钮" : Bool;
      "3层上行呼梯按钮" : Bool;
      "4层上行呼梯按钮" : Bool;
      "5层上行呼梯按钮" : Bool;
      "6层上行呼梯按钮" : Bool;
      "7层上行呼梯按钮" : Bool;
      "8层上行呼梯按钮" : Bool;
      "9层上行呼梯按钮" : Bool;
      "2层下行呼梯按钮" : Bool;
      "3层下行呼梯按钮" : Bool;
      "4层下行呼梯按钮" : Bool;
      "5层下行呼梯按钮" : Bool;
      "6层下行呼梯按钮" : Bool;
      "7层下行呼梯按钮" : Bool;
      "8层下行呼梯按钮" : Bool;
      "9层下行呼梯按钮" : Bool;
      "10层下行呼梯按钮" : Bool;
      "1号梯轿内选层按钮1" : Bool;
      "1号梯轿内选层按钮2" : Bool;
      "1号梯轿内选层按钮3" : Bool;
      "1号梯轿内选层按钮4" : Bool;
      "1号梯轿内选层按钮5" : Bool;
      "1号梯轿内选层按钮6" : Bool;
      "1号梯轿内选层按钮7" : Bool;
      "1号梯轿内选层按钮8" : Bool;
      "1号梯轿内选层按钮9" : Bool;
      "1号梯轿内选层按钮10" : Bool;
      "1号梯轿内开门按钮" : Bool;
      "1号梯轿内关门按钮" : Bool;
      "1号梯光幕信号" : Bool;
      "1号梯检修信号" : Bool;
      "1号梯轿厢门锁信号" : Bool;
      "1号梯1楼层门锁信号" : Bool;
      "1号梯2楼层门锁信号" : Bool;
      "1号梯3楼层门锁信号" : Bool;
      "1号梯4楼层门锁信号" : Bool;
      "1号梯5楼层门锁信号" : Bool;
      "1号梯6楼层门锁信号" : Bool;
      "1号梯7楼层门锁信号" : Bool;
      "1号梯8楼层门锁信号" : Bool;
      "1号梯9楼层门锁信号" : Bool;
      "1号梯10楼层门锁信号" : Bool;
      "1号梯开门到位" : Bool;
      "1号梯关门到位" : Bool;
      "1号梯上平层信号" : Bool;
      "1号梯下平层信号" : Bool;
      "1号梯上端站第1限位" : Bool;
      "1号梯上端站第2限位" : Bool;
      "1号梯下端站第1限位" : Bool;
      "1号梯下端站第2限位" : Bool;
      "2号梯轿内选层按钮1" : Bool;
      "2号梯轿内选层按钮2" : Bool;
      "2号梯轿内选层按钮3" : Bool;
      "2号梯轿内选层按钮4" : Bool;
      "2号梯轿内选层按钮5" : Bool;
      "2号梯轿内选层按钮6" : Bool;
      "2号梯轿内选层按钮7" : Bool;
      "2号梯轿内选层按钮8" : Bool;
      "2号梯轿内选层按钮9" : Bool;
      "2号梯轿内选层按钮10" : Bool;
      "2号梯轿内开门按钮" : Bool;
      "2号梯轿内关门按钮" : Bool;
      "2号梯光幕信号" : Bool;
      "2号梯检修信号" : Bool;
      "2号梯轿厢门锁信号" : Bool;
      "2号梯1楼层门锁信号" : Bool;
      "2号梯2楼层门锁信号" : Bool;
      "2号梯3楼层门锁信号" : Bool;
      "2号梯4楼层门锁信号" : Bool;
      "2号梯5楼层门锁信号" : Bool;
      "2号梯6楼层门锁信号" : Bool;
      "2号梯7楼层门锁信号" : Bool;
      "2号梯8楼层门锁信号" : Bool;
      "2号梯9楼层门锁信号" : Bool;
      "2号梯10楼层门锁信号" : Bool;
      "2号梯开门到位" : Bool;
      "2号梯关门到位" : Bool;
      "2号梯上平层信号" : Bool;
      "2号梯下平层信号" : Bool;
      "2号梯上端站第1限位" : Bool;
      "2号梯上端站第2限位" : Bool;
      "2号梯下端站第1限位" : Bool;
      "2号梯下端站第2限位" : Bool;
      "3号梯轿内选层按钮1" : Bool;
      "3号梯轿内选层按钮2" : Bool;
      "3号梯轿内选层按钮3" : Bool;
      "3号梯轿内选层按钮4" : Bool;
      "3号梯轿内选层按钮5" : Bool;
      "3号梯轿内选层按钮6" : Bool;
      "3号梯轿内选层按钮7" : Bool;
      "3号梯轿内选层按钮8" : Bool;
      "3号梯轿内选层按钮9" : Bool;
      "3号梯轿内选层按钮10" : Bool;
      "3号梯轿内开门按钮" : Bool;
      "3号梯轿内关门按钮" : Bool;
      "3号梯光幕信号" : Bool;
      "3号梯检修信号" : Bool;
      "3号梯轿厢门锁信号" : Bool;
      "3号梯1楼层门锁信号" : Bool;
      "3号梯2楼层门锁信号" : Bool;
      "3号梯3楼层门锁信号" : Bool;
      "3号梯4楼层门锁信号" : Bool;
      "3号梯5楼层门锁信号" : Bool;
      "3号梯6楼层门锁信号" : Bool;
      "3号梯7楼层门锁信号" : Bool;
      "3号梯8楼层门锁信号" : Bool;
      "3号梯9楼层门锁信号" : Bool;
      "3号梯10楼层门锁信号" : Bool;
      "3号梯开门到位" : Bool;
      "3号梯关门到位" : Bool;
      "3号梯上平层信号" : Bool;
      "3号梯下平层信号" : Bool;
      "3号梯上端站第1限位" : Bool;
      "3号梯上端站第2限位" : Bool;
      "3号梯下端站第1限位" : Bool;
      "3号梯下端站第2限位" : Bool;
      自动运行信号 : Bool;
      "1号梯当前载重量" : Word;
      "2号梯当前载重量" : Word;
      "3号梯当前载重量" : Word;
   END_VAR
BEGIN
END_DATA_BLOCK

DATA_BLOCK "output"   // DB11
{ S7_Optimized_Access := 'FALSE' }
VERSION : 0.1
   VAR
      "1层上行呼梯按钮指示灯" : Bool;
      "2层上行呼梯按钮指示灯" : Bool;
      "3层上行呼梯按钮指示灯" : Bool;
      "4层上行呼梯按钮指示灯" : Bool;
      "5层上行呼梯按钮指示灯" : Bool;
      "6层上行呼梯按钮指示灯" : Bool;
      "7层上行呼梯按钮指示灯" : Bool;
      "8层上行呼梯按钮指示灯" : Bool;
      "9层上行呼梯按钮指示灯" : Bool;
      "2层下行呼梯按钮指示灯" : Bool;
      "3层下行呼梯按钮指示灯" : Bool;
      "4层下行呼梯按钮指示灯" : Bool;
      "5层下行呼梯按钮指示灯" : Bool;
      "6层下行呼梯按钮指示灯" : Bool;
      "7层下行呼梯按钮指示灯" : Bool;
      "8层下行呼梯按钮指示灯" : Bool;
      "9层下行呼梯按钮指示灯" : Bool;
      "10层下行呼梯按钮指示灯" : Bool;
      "1号梯1层按钮指示灯" : Bool;
      "1号梯2层按钮指示灯" : Bool;
      "1号梯3层按钮指示灯" : Bool;
      "1号梯4层按钮指示灯" : Bool;
      "1号梯5层按钮指示灯" : Bool;
      "1号梯6层按钮指示灯" : Bool;
      "1号梯7层按钮指示灯" : Bool;
      "1号梯8层按钮指示灯" : Bool;
      "1号梯9层按钮指示灯" : Bool;
      "1号梯10层按钮指示灯" : Bool;
      "1号梯LEDa" : Bool;
      "1号梯LEDb" : Bool;
      "1号梯LEDc" : Bool;
      "1号梯LEDd" : Bool;
      "1号梯LEDe" : Bool;
      "1号梯LEDf" : Bool;
      "1号梯LEDg" : Bool;
      "1号梯LEDh" : Bool;
      "1号梯LEDi" : Bool;
      "1号梯LEDj" : Bool;
      "1号梯LEDk" : Bool;
      "1号梯LEDl" : Bool;
      "1号梯LEDm" : Bool;
      "1号梯LEDn" : Bool;
      "1号梯上行指示" : Bool;
      "1号梯下行指示" : Bool;
      "1号梯故障指示" : Bool;
      "1号梯照明指示" : Bool;
      "1号梯风扇指示" : Bool;
      "1号梯满载指示" : Bool;
      "1号梯电机启动信号" : Bool;
      "1号梯上行接触器" : Bool;
      "1号梯下行接触器" : Bool;
      "1号梯高速接触器" : Bool;
      "1号梯低速接触器" : Bool;
      "1号梯开门继电器" : Bool;
      "1号梯关门继电器" : Bool;
      "1号梯1级减速制动" : Bool;
      "1号梯2级减速制动" : Bool;
      "1号梯3级减速制动" : Bool;
      "2号梯1层按钮指示灯" : Bool;
      "2号梯2层按钮指示灯" : Bool;
      "2号梯3层按钮指示灯" : Bool;
      "2号梯4层按钮指示灯" : Bool;
      "2号梯5层按钮指示灯" : Bool;
      "2号梯6层按钮指示灯" : Bool;
      "2号梯7层按钮指示灯" : Bool;
      "2号梯8层按钮指示灯" : Bool;
      "2号梯9层按钮指示灯" : Bool;
      "2号梯10层按钮指示灯" : Bool;
      "2号梯LEDa" : Bool;
      "2号梯LEDb" : Bool;
      "2号梯LEDc" : Bool;
      "2号梯LEDd" : Bool;
      "2号梯LEDe" : Bool;
      "2号梯LEDf" : Bool;
      "2号梯LEDg" : Bool;
      "2号梯LEDh" : Bool;
      "2号梯LEDi" : Bool;
      "2号梯LEDj" : Bool;
      "2号梯LEDk" : Bool;
      "2号梯LEDl" : Bool;
      "2号梯LEDm" : Bool;
      "2号梯LEDn" : Bool;
      "2号梯上行指示" : Bool;
      "2号梯下行指示" : Bool;
      "2号梯故障指示" : Bool;
      "2号梯照明指示" : Bool;
      "2号梯风扇指示" : Bool;
      "2号梯满载指示" : Bool;
      "2号梯电机启动信号" : Bool;
      "2号梯上行接触器" : Bool;
      "2号梯下行接触器" : Bool;
      "2号梯高速接触器" : Bool;
      "2号梯低速接触器" : Bool;
      "2号梯开门继电器" : Bool;
      "2号梯关门继电器" : Bool;
      "2号梯1级减速制动" : Bool;
      "2号梯2级减速制动" : Bool;
      "2号梯3级减速制动" : Bool;
      "3号梯1层按钮指示灯" : Bool;
      "3号梯2层按钮指示灯" : Bool;
      "3号梯3层按钮指示灯" : Bool;
      "3号梯4层按钮指示灯" : Bool;
      "3号梯5层按钮指示灯" : Bool;
      "3号梯6层按钮指示灯" : Bool;
      "3号梯7层按钮指示灯" : Bool;
      "3号梯8层按钮指示灯" : Bool;
      "3号梯9层按钮指示灯" : Bool;
      "3号梯10层按钮指示灯" : Bool;
      "3号梯LEDa" : Bool;
      "3号梯LEDb" : Bool;
      "3号梯LEDc" : Bool;
      "3号梯LEDd" : Bool;
      "3号梯LEDe" : Bool;
      "3号梯LEDf" : Bool;
      "3号梯LEDg" : Bool;
      "3号梯LEDh" : Bool;
      "3号梯LEDi" : Bool;
      "3号梯LEDj" : Bool;
      "3号梯LEDk" : Bool;
      "3号梯LEDl" : Bool;
      "3号梯LEDm" : Bool;
      "3号梯LEDn" : Bool;
      "3号梯上行指示" : Bool;
      "3号梯下行指示" : Bool;
      "3号梯故障指示" : Bool;
      "3号梯照明指示" : Bool;
      "3号梯风扇指示" : Bool;
      "3号梯满载指示" : Bool;
      "3号梯电机启动信号" : Bool;
      "3号梯上行接触器" : Bool;
      "3号梯下行接触器" : Bool;
      "3号梯高速接触器" : Bool;
      "3号梯低速接触器" : Bool;
      "3号梯开门继电器" : Bool;
      "3号梯关门继电器" : Bool;
      "3号梯1级减速制动" : Bool;
      "3号梯2级减速制动" : Bool;
      "3号梯3级减速制动" : Bool;
      准备就绪信号 : Bool;
   END_VAR
BEGIN
END_DATA_BLOCK

DATA_BLOCK "DB_GC"   // DB51
{ S7_Optimized_Access := 'FALSE' }
VERSION : 0.1
   VAR
      HallUpBtn : Array[1..10] of Bool;
      HallDownBtn : Array[1..10] of Bool;
      LiftCarCall : Array[1..3, 1..10] of Bool;
      LiftHallUp : Array[1..3, 1..10] of Bool;
      LiftHallDown : Array[1..3, 1..10] of Bool;
      LiftFloor : Array[1..3] of Int;   // 当前楼层
      LiftDir : Array[1..3] of Int;   // 运行方向
      LiftRunning : Array[1..3] of Bool;   // 运行状态
      LiftDoorOpen : Array[1..3] of Bool;   // 开门状态
      LiftLoadPercent : Array[1..3] of Int;   // 载客率
      LiftPower_kW : Array[1..3] of Real;   // 功率
      LiftGroupEnable : Array[1..3] of Bool;   // 群控使能
      LiftLocked : Array[1..3] of Bool;   // 锁梯
      LiftDisabled : Array[1..3] of Bool;   // 禁用
      GroupMode : Int;   // 模式
      RideFinishPulse : Array[1..3] of Bool;   // 乘梯
      RideTimeSample_s : Array[1..3] of Real;
      AssignedLiftUp : Array[1..10] of Int;
      AssignedLiftDown : Array[1..10] of Int;
      LiftTaskCount : Array[1..3] of Int;
      AheadTaskCountOut : Array[1..3] of Int;
      AvgWait_s : Real;
      CurrentAvgWait_s : Real;
      CurrentWaitingCount : Int;
      LongWaitRatePercent : Real;
      AvgRideTime_s : Real;
      LiftEfficiencyPercent : Array[1..3] of Real;
      SystemEmptyRatePercent : Real;
      LiftEnergy_kWh : Array[1..3] of Real;
      SystemEnergy_kWh : Real;
      HallUpLampOut : Array[1..10] of Bool;
      HallDownLampOut : Array[1..10] of Bool;
      HallUpCancel : Array[1..10] of Bool;
      HallDownCancel : Array[1..10] of Bool;
   END_VAR
BEGIN
END_DATA_BLOCK

DATA_BLOCK "FB_GC_3Lift_10Floor_DB_1"   // DB83
{ S7_Optimized_Access := 'TRUE' }
VERSION : 0.1
// stored: InstanceOfName FB_GC_3Lift_10Floor
"FB_GC_3Lift_10Floor"
BEGIN
   CycleTime_s := 0.1;
   LongWaitLimit_s := 60.0;
   FullLoadLimitPercent := 95;
   EmptyLoadLimitPercent := 15;
   W_Distance := 10;
   W_Direction := 30;
   W_Task := 15;
   W_AheadTask := 15;
   W_LoadPercent := 0.2;
   empty := 40;
END_DATA_BLOCK

// folder: System blocks/Program resources

DATA_BLOCK "IEC_Timer_0_DB"   // DB1
{ S7_Optimized_Access := 'TRUE' }
AUTHOR : Simatic
FAMILY : IEC
NAME : IEC_TMR
VERSION : 1.0
// stored: InstanceOfName IEC_TIMER
"IEC_TIMER"
BEGIN
END_DATA_BLOCK

DATA_BLOCK "IEC_Timer_0_DB_1"   // DB2
{ S7_Optimized_Access := 'TRUE' }
AUTHOR : Simatic
FAMILY : IEC
NAME : IEC_TMR
VERSION : 1.0
// stored: InstanceOfName IEC_TIMER
"IEC_TIMER"
BEGIN
END_DATA_BLOCK

DATA_BLOCK "IEC_Timer_0_DB_2"   // DB3
{ S7_Optimized_Access := 'TRUE' }
AUTHOR : Simatic
FAMILY : IEC
NAME : IEC_TMR
VERSION : 1.0
// stored: InstanceOfName IEC_TIMER
"IEC_TIMER"
BEGIN
END_DATA_BLOCK

DATA_BLOCK "T1"   // DB4
{ S7_Optimized_Access := 'TRUE' }
AUTHOR : Simatic
FAMILY : IEC
NAME : IEC_TMR
VERSION : 1.0
// stored: InstanceOfName IEC_TIMER
"IEC_TIMER"
BEGIN
END_DATA_BLOCK

DATA_BLOCK "T2"   // DB5
{ S7_Optimized_Access := 'TRUE' }
AUTHOR : Simatic
FAMILY : IEC
NAME : IEC_TMR
VERSION : 1.0
// stored: InstanceOfName IEC_TIMER
"IEC_TIMER"
BEGIN
END_DATA_BLOCK

DATA_BLOCK "T3"   // DB6
{ S7_Optimized_Access := 'TRUE' }
AUTHOR : Simatic
FAMILY : IEC
NAME : IEC_TMR
VERSION : 1.0
// stored: InstanceOfName IEC_TIMER
"IEC_TIMER"
BEGIN
END_DATA_BLOCK

DATA_BLOCK "IEC_Timer_0_DB_3"   // DB7
{ S7_Optimized_Access := 'TRUE' }
AUTHOR : Simatic
FAMILY : IEC
NAME : IEC_TMR
VERSION : 1.0
// stored: InstanceOfName IEC_TIMER
"IEC_TIMER"
BEGIN
END_DATA_BLOCK

DATA_BLOCK "IEC_Timer_0_DB_5"   // DB8
{ S7_Optimized_Access := 'TRUE' }
AUTHOR : Simatic
FAMILY : IEC
NAME : IEC_TMR
VERSION : 1.0
// stored: InstanceOfName IEC_TIMER
"IEC_TIMER"
BEGIN
END_DATA_BLOCK

DATA_BLOCK "IEC_Timer_0_DB_4"   // DB9
{ S7_Optimized_Access := 'TRUE' }
AUTHOR : Simatic
FAMILY : IEC
NAME : IEC_TMR
VERSION : 1.0
// stored: InstanceOfName IEC_TIMER
"IEC_TIMER"
BEGIN
END_DATA_BLOCK

DATA_BLOCK "IEC_Timer_0_DB_6"   // DB12
{ S7_Optimized_Access := 'TRUE' }
AUTHOR : Simatic
FAMILY : IEC
NAME : IEC_TMR
VERSION : 1.0
// stored: InstanceOfName IEC_TIMER
"IEC_TIMER"
BEGIN
END_DATA_BLOCK

DATA_BLOCK "IEC_Timer_0_DB_7"   // DB13
{ S7_Optimized_Access := 'TRUE' }
AUTHOR : Simatic
FAMILY : IEC
NAME : IEC_TMR
VERSION : 1.0
// stored: InstanceOfName IEC_TIMER
"IEC_TIMER"
BEGIN
END_DATA_BLOCK

DATA_BLOCK "IEC_Timer_0_DB_8"   // DB14
{ S7_Optimized_Access := 'TRUE' }
AUTHOR : Simatic
FAMILY : IEC
NAME : IEC_TMR
VERSION : 1.0
// stored: InstanceOfName IEC_TIMER
"IEC_TIMER"
BEGIN
END_DATA_BLOCK

DATA_BLOCK "IEC_Timer_0_DB_9"   // DB15
{ S7_Optimized_Access := 'TRUE' }
AUTHOR : Simatic
FAMILY : IEC
NAME : IEC_TMR
VERSION : 1.0
// stored: InstanceOfName IEC_TIMER
"IEC_TIMER"
BEGIN
END_DATA_BLOCK

DATA_BLOCK "IEC_Timer_0_DB_10"   // DB16
{ S7_Optimized_Access := 'TRUE' }
AUTHOR : Simatic
FAMILY : IEC
NAME : IEC_TMR
VERSION : 1.0
// stored: InstanceOfName IEC_TIMER
"IEC_TIMER"
BEGIN
END_DATA_BLOCK

DATA_BLOCK "IEC_Timer_0_DB_11"   // DB17
{ S7_Optimized_Access := 'TRUE' }
AUTHOR : Simatic
FAMILY : IEC
NAME : IEC_TMR
VERSION : 1.0
// stored: InstanceOfName IEC_TIMER
"IEC_TIMER"
BEGIN
END_DATA_BLOCK

DATA_BLOCK "IEC_Timer_0_DB_18"   // DB18
{ S7_Optimized_Access := 'TRUE' }
AUTHOR : Simatic
FAMILY : IEC
NAME : IEC_TMR
VERSION : 1.0
// stored: InstanceOfName IEC_TIMER
"IEC_TIMER"
BEGIN
END_DATA_BLOCK

DATA_BLOCK "IEC_Timer_0_DB_19"   // DB19
{ S7_Optimized_Access := 'TRUE' }
AUTHOR : Simatic
FAMILY : IEC
NAME : IEC_TMR
VERSION : 1.0
// stored: InstanceOfName IEC_TIMER
"IEC_TIMER"
BEGIN
END_DATA_BLOCK

DATA_BLOCK "IEC_Timer_0_DB_20"   // DB20
{ S7_Optimized_Access := 'TRUE' }
AUTHOR : Simatic
FAMILY : IEC
NAME : IEC_TMR
VERSION : 1.0
// stored: InstanceOfName IEC_TIMER
"IEC_TIMER"
BEGIN
END_DATA_BLOCK

DATA_BLOCK "IEC_Timer_0_DB_21"   // DB21
{ S7_Optimized_Access := 'TRUE' }
AUTHOR : Simatic
FAMILY : IEC
NAME : IEC_TMR
VERSION : 1.0
// stored: InstanceOfName IEC_TIMER
"IEC_TIMER"
BEGIN
END_DATA_BLOCK

DATA_BLOCK "IEC_Timer_0_DB_22"   // DB22
{ S7_Optimized_Access := 'TRUE' }
AUTHOR : Simatic
FAMILY : IEC
NAME : IEC_TMR
VERSION : 1.0
// stored: InstanceOfName IEC_TIMER
"IEC_TIMER"
BEGIN
END_DATA_BLOCK

DATA_BLOCK "IEC_Timer_0_DB_23"   // DB23
{ S7_Optimized_Access := 'TRUE' }
AUTHOR : Simatic
FAMILY : IEC
NAME : IEC_TMR
VERSION : 1.0
// stored: InstanceOfName IEC_TIMER
"IEC_TIMER"
BEGIN
END_DATA_BLOCK

DATA_BLOCK "IEC_Timer_0_DB_24"   // DB24
{ S7_Optimized_Access := 'TRUE' }
AUTHOR : Simatic
FAMILY : IEC
NAME : IEC_TMR
VERSION : 1.0
// stored: InstanceOfName IEC_TIMER
"IEC_TIMER"
BEGIN
END_DATA_BLOCK

DATA_BLOCK "IEC_Timer_0_DB_30"   // DB25
{ S7_Optimized_Access := 'TRUE' }
AUTHOR : Simatic
FAMILY : IEC
NAME : IEC_TMR
VERSION : 1.0
// stored: InstanceOfName IEC_TIMER
"IEC_TIMER"
BEGIN
END_DATA_BLOCK

DATA_BLOCK "IEC_Timer_0_DB_12"   // DB26
{ S7_Optimized_Access := 'TRUE' }
AUTHOR : Simatic
FAMILY : IEC
NAME : IEC_TMR
VERSION : 1.0
// stored: InstanceOfName IEC_TIMER
"IEC_TIMER"
BEGIN
END_DATA_BLOCK

DATA_BLOCK "IEC_Timer_0_DB_13"   // DB27
{ S7_Optimized_Access := 'TRUE' }
AUTHOR : Simatic
FAMILY : IEC
NAME : IEC_TMR
VERSION : 1.0
// stored: InstanceOfName IEC_TIMER
"IEC_TIMER"
BEGIN
END_DATA_BLOCK

DATA_BLOCK "IEC_Timer_0_DB_14"   // DB28
{ S7_Optimized_Access := 'TRUE' }
AUTHOR : Simatic
FAMILY : IEC
NAME : IEC_TMR
VERSION : 1.0
// stored: InstanceOfName IEC_TIMER
"IEC_TIMER"
BEGIN
END_DATA_BLOCK

DATA_BLOCK "IEC_Timer_0_DB_15"   // DB29
{ S7_Optimized_Access := 'TRUE' }
AUTHOR : Simatic
FAMILY : IEC
NAME : IEC_TMR
VERSION : 1.0
// stored: InstanceOfName IEC_TIMER
"IEC_TIMER"
BEGIN
END_DATA_BLOCK

DATA_BLOCK "IEC_Timer_0_DB_16"   // DB30
{ S7_Optimized_Access := 'TRUE' }
AUTHOR : Simatic
FAMILY : IEC
NAME : IEC_TMR
VERSION : 1.0
// stored: InstanceOfName IEC_TIMER
"IEC_TIMER"
BEGIN
END_DATA_BLOCK

DATA_BLOCK "IEC_Timer_0_DB_17"   // DB31
{ S7_Optimized_Access := 'TRUE' }
AUTHOR : Simatic
FAMILY : IEC
NAME : IEC_TMR
VERSION : 1.0
// stored: InstanceOfName IEC_TIMER
"IEC_TIMER"
BEGIN
END_DATA_BLOCK

DATA_BLOCK "IEC_Timer_0_DB_31"   // DB32
{ S7_Optimized_Access := 'TRUE' }
AUTHOR : Simatic
FAMILY : IEC
NAME : IEC_TMR
VERSION : 1.0
// stored: InstanceOfName IEC_TIMER
"IEC_TIMER"
BEGIN
END_DATA_BLOCK

DATA_BLOCK "IEC_Timer_0_DB_32"   // DB33
{ S7_Optimized_Access := 'TRUE' }
AUTHOR : Simatic
FAMILY : IEC
NAME : IEC_TMR
VERSION : 1.0
// stored: InstanceOfName IEC_TIMER
"IEC_TIMER"
BEGIN
END_DATA_BLOCK

DATA_BLOCK "IEC_Timer_0_DB_33"   // DB34
{ S7_Optimized_Access := 'TRUE' }
AUTHOR : Simatic
FAMILY : IEC
NAME : IEC_TMR
VERSION : 1.0
// stored: InstanceOfName IEC_TIMER
"IEC_TIMER"
BEGIN
END_DATA_BLOCK

DATA_BLOCK "IEC_Timer_0_DB_34"   // DB35
{ S7_Optimized_Access := 'TRUE' }
AUTHOR : Simatic
FAMILY : IEC
NAME : IEC_TMR
VERSION : 1.0
// stored: InstanceOfName IEC_TIMER
"IEC_TIMER"
BEGIN
END_DATA_BLOCK

DATA_BLOCK "IEC_Timer_0_DB_35"   // DB36
{ S7_Optimized_Access := 'TRUE' }
AUTHOR : Simatic
FAMILY : IEC
NAME : IEC_TMR
VERSION : 1.0
// stored: InstanceOfName IEC_TIMER
"IEC_TIMER"
BEGIN
END_DATA_BLOCK

DATA_BLOCK "IEC_Timer_0_DB_36"   // DB37
{ S7_Optimized_Access := 'TRUE' }
AUTHOR : Simatic
FAMILY : IEC
NAME : IEC_TMR
VERSION : 1.0
// stored: InstanceOfName IEC_TIMER
"IEC_TIMER"
BEGIN
END_DATA_BLOCK

DATA_BLOCK "IEC_Timer_0_DB_37"   // DB38
{ S7_Optimized_Access := 'TRUE' }
AUTHOR : Simatic
FAMILY : IEC
NAME : IEC_TMR
VERSION : 1.0
// stored: InstanceOfName IEC_TIMER
"IEC_TIMER"
BEGIN
END_DATA_BLOCK

DATA_BLOCK "IEC_Timer_0_DB_38"   // DB39
{ S7_Optimized_Access := 'TRUE' }
AUTHOR : Simatic
FAMILY : IEC
NAME : IEC_TMR
VERSION : 1.0
// stored: InstanceOfName IEC_TIMER
"IEC_TIMER"
BEGIN
END_DATA_BLOCK

DATA_BLOCK "IEC_Timer_0_DB_39"   // DB40
{ S7_Optimized_Access := 'TRUE' }
AUTHOR : Simatic
FAMILY : IEC
NAME : IEC_TMR
VERSION : 1.0
// stored: InstanceOfName IEC_TIMER
"IEC_TIMER"
BEGIN
END_DATA_BLOCK

DATA_BLOCK "IEC_Timer_0_DB_25"   // DB41
{ S7_Optimized_Access := 'TRUE' }
AUTHOR : Simatic
FAMILY : IEC
NAME : IEC_TMR
VERSION : 1.0
// stored: InstanceOfName IEC_TIMER
"IEC_TIMER"
BEGIN
END_DATA_BLOCK

DATA_BLOCK "IEC_Timer_0_DB_26"   // DB42
{ S7_Optimized_Access := 'TRUE' }
AUTHOR : Simatic
FAMILY : IEC
NAME : IEC_TMR
VERSION : 1.0
// stored: InstanceOfName IEC_TIMER
"IEC_TIMER"
BEGIN
END_DATA_BLOCK

DATA_BLOCK "IEC_Timer_0_DB_27"   // DB43
{ S7_Optimized_Access := 'TRUE' }
AUTHOR : Simatic
FAMILY : IEC
NAME : IEC_TMR
VERSION : 1.0
// stored: InstanceOfName IEC_TIMER
"IEC_TIMER"
BEGIN
END_DATA_BLOCK

DATA_BLOCK "IEC_Timer_0_DB_28"   // DB44
{ S7_Optimized_Access := 'TRUE' }
AUTHOR : Simatic
FAMILY : IEC
NAME : IEC_TMR
VERSION : 1.0
// stored: InstanceOfName IEC_TIMER
"IEC_TIMER"
BEGIN
END_DATA_BLOCK

DATA_BLOCK "IEC_Timer_0_DB_29"   // DB45
{ S7_Optimized_Access := 'TRUE' }
AUTHOR : Simatic
FAMILY : IEC
NAME : IEC_TMR
VERSION : 1.0
// stored: InstanceOfName IEC_TIMER
"IEC_TIMER"
BEGIN
END_DATA_BLOCK

DATA_BLOCK "IEC_Timer_0_DB_40"   // DB46
{ S7_Optimized_Access := 'TRUE' }
AUTHOR : Simatic
FAMILY : IEC
NAME : IEC_TMR
VERSION : 1.0
// stored: InstanceOfName IEC_TIMER
"IEC_TIMER"
BEGIN
END_DATA_BLOCK

DATA_BLOCK "IEC_Timer_0_DB_41"   // DB47
{ S7_Optimized_Access := 'TRUE' }
AUTHOR : Simatic
FAMILY : IEC
NAME : IEC_TMR
VERSION : 1.0
// stored: InstanceOfName IEC_TIMER
"IEC_TIMER"
BEGIN
END_DATA_BLOCK

DATA_BLOCK "IEC_Timer_0_DB_42"   // DB48
{ S7_Optimized_Access := 'TRUE' }
AUTHOR : Simatic
FAMILY : IEC
NAME : IEC_TMR
VERSION : 1.0
// stored: InstanceOfName IEC_TIMER
"IEC_TIMER"
BEGIN
END_DATA_BLOCK

DATA_BLOCK "IEC_Timer_0_DB_43"   // DB49
{ S7_Optimized_Access := 'TRUE' }
AUTHOR : Simatic
FAMILY : IEC
NAME : IEC_TMR
VERSION : 1.0
// stored: InstanceOfName IEC_TIMER
"IEC_TIMER"
BEGIN
END_DATA_BLOCK

DATA_BLOCK "IEC_Timer_0_DB_44"   // DB50
{ S7_Optimized_Access := 'TRUE' }
AUTHOR : Simatic
FAMILY : IEC
NAME : IEC_TMR
VERSION : 1.0
// stored: InstanceOfName IEC_TIMER
"IEC_TIMER"
BEGIN
END_DATA_BLOCK

DATA_BLOCK "IEC_Timer_0_DB_105"   // DB52
{ S7_Optimized_Access := 'TRUE' }
AUTHOR : Simatic
FAMILY : IEC
NAME : IEC_TMR
VERSION : 1.0
// stored: InstanceOfName IEC_TIMER
"IEC_TIMER"
BEGIN
END_DATA_BLOCK

DATA_BLOCK "IEC_Timer_0_DB_60"   // DB53
{ S7_Optimized_Access := 'TRUE' }
AUTHOR : Simatic
FAMILY : IEC
NAME : IEC_TMR
VERSION : 1.0
// stored: InstanceOfName IEC_TIMER
"IEC_TIMER"
BEGIN
END_DATA_BLOCK

DATA_BLOCK "IEC_Timer_0_DB_61"   // DB54
{ S7_Optimized_Access := 'TRUE' }
AUTHOR : Simatic
FAMILY : IEC
NAME : IEC_TMR
VERSION : 1.0
// stored: InstanceOfName IEC_TIMER
"IEC_TIMER"
BEGIN
END_DATA_BLOCK

DATA_BLOCK "IEC_Timer_0_DB_46"   // DB55
{ S7_Optimized_Access := 'TRUE' }
AUTHOR : Simatic
FAMILY : IEC
NAME : IEC_TMR
VERSION : 1.0
// stored: InstanceOfName IEC_TIMER
"IEC_TIMER"
BEGIN
END_DATA_BLOCK

DATA_BLOCK "IEC_Timer_0_DB_47"   // DB56
{ S7_Optimized_Access := 'TRUE' }
AUTHOR : Simatic
FAMILY : IEC
NAME : IEC_TMR
VERSION : 1.0
// stored: InstanceOfName IEC_TIMER
"IEC_TIMER"
BEGIN
END_DATA_BLOCK

DATA_BLOCK "IEC_Timer_0_DB_48"   // DB57
{ S7_Optimized_Access := 'TRUE' }
AUTHOR : Simatic
FAMILY : IEC
NAME : IEC_TMR
VERSION : 1.0
// stored: InstanceOfName IEC_TIMER
"IEC_TIMER"
BEGIN
END_DATA_BLOCK

DATA_BLOCK "IEC_Timer_0_DB_49"   // DB58
{ S7_Optimized_Access := 'TRUE' }
AUTHOR : Simatic
FAMILY : IEC
NAME : IEC_TMR
VERSION : 1.0
// stored: InstanceOfName IEC_TIMER
"IEC_TIMER"
BEGIN
END_DATA_BLOCK

DATA_BLOCK "IEC_Timer_0_DB_62"   // DB59
{ S7_Optimized_Access := 'TRUE' }
AUTHOR : Simatic
FAMILY : IEC
NAME : IEC_TMR
VERSION : 1.0
// stored: InstanceOfName IEC_TIMER
"IEC_TIMER"
BEGIN
END_DATA_BLOCK

DATA_BLOCK "IEC_Timer_0_DB_63"   // DB60
{ S7_Optimized_Access := 'TRUE' }
AUTHOR : Simatic
FAMILY : IEC
NAME : IEC_TMR
VERSION : 1.0
// stored: InstanceOfName IEC_TIMER
"IEC_TIMER"
BEGIN
END_DATA_BLOCK

DATA_BLOCK "IEC_Timer_0_DB_64"   // DB61
{ S7_Optimized_Access := 'TRUE' }
AUTHOR : Simatic
FAMILY : IEC
NAME : IEC_TMR
VERSION : 1.0
// stored: InstanceOfName IEC_TIMER
"IEC_TIMER"
BEGIN
END_DATA_BLOCK

DATA_BLOCK "IEC_Timer_0_DB_65"   // DB62
{ S7_Optimized_Access := 'TRUE' }
AUTHOR : Simatic
FAMILY : IEC
NAME : IEC_TMR
VERSION : 1.0
// stored: InstanceOfName IEC_TIMER
"IEC_TIMER"
BEGIN
END_DATA_BLOCK

DATA_BLOCK "IEC_Timer_0_DB_50"   // DB63
{ S7_Optimized_Access := 'TRUE' }
AUTHOR : Simatic
FAMILY : IEC
NAME : IEC_TMR
VERSION : 1.0
// stored: InstanceOfName IEC_TIMER
"IEC_TIMER"
BEGIN
END_DATA_BLOCK

DATA_BLOCK "IEC_Timer_0_DB_66"   // DB64
{ S7_Optimized_Access := 'TRUE' }
AUTHOR : Simatic
FAMILY : IEC
NAME : IEC_TMR
VERSION : 1.0
// stored: InstanceOfName IEC_TIMER
"IEC_TIMER"
BEGIN
END_DATA_BLOCK

DATA_BLOCK "IEC_Timer_0_DB_51"   // DB65
{ S7_Optimized_Access := 'TRUE' }
AUTHOR : Simatic
FAMILY : IEC
NAME : IEC_TMR
VERSION : 1.0
// stored: InstanceOfName IEC_TIMER
"IEC_TIMER"
BEGIN
END_DATA_BLOCK

DATA_BLOCK "IEC_Timer_0_DB_67"   // DB66
{ S7_Optimized_Access := 'TRUE' }
AUTHOR : Simatic
FAMILY : IEC
NAME : IEC_TMR
VERSION : 1.0
// stored: InstanceOfName IEC_TIMER
"IEC_TIMER"
BEGIN
END_DATA_BLOCK

DATA_BLOCK "IEC_Timer_0_DB_52"   // DB67
{ S7_Optimized_Access := 'TRUE' }
AUTHOR : Simatic
FAMILY : IEC
NAME : IEC_TMR
VERSION : 1.0
// stored: InstanceOfName IEC_TIMER
"IEC_TIMER"
BEGIN
END_DATA_BLOCK

DATA_BLOCK "IEC_Timer_0_DB_68"   // DB68
{ S7_Optimized_Access := 'TRUE' }
AUTHOR : Simatic
FAMILY : IEC
NAME : IEC_TMR
VERSION : 1.0
// stored: InstanceOfName IEC_TIMER
"IEC_TIMER"
BEGIN
END_DATA_BLOCK

DATA_BLOCK "IEC_Timer_0_DB_53"   // DB69
{ S7_Optimized_Access := 'TRUE' }
AUTHOR : Simatic
FAMILY : IEC
NAME : IEC_TMR
VERSION : 1.0
// stored: InstanceOfName IEC_TIMER
"IEC_TIMER"
BEGIN
END_DATA_BLOCK

DATA_BLOCK "IEC_Timer_0_DB_69"   // DB70
{ S7_Optimized_Access := 'TRUE' }
AUTHOR : Simatic
FAMILY : IEC
NAME : IEC_TMR
VERSION : 1.0
// stored: InstanceOfName IEC_TIMER
"IEC_TIMER"
BEGIN
END_DATA_BLOCK

DATA_BLOCK "IEC_Timer_0_DB_54"   // DB71
{ S7_Optimized_Access := 'TRUE' }
AUTHOR : Simatic
FAMILY : IEC
NAME : IEC_TMR
VERSION : 1.0
// stored: InstanceOfName IEC_TIMER
"IEC_TIMER"
BEGIN
END_DATA_BLOCK

DATA_BLOCK "IEC_Timer_0_DB_70"   // DB72
{ S7_Optimized_Access := 'TRUE' }
AUTHOR : Simatic
FAMILY : IEC
NAME : IEC_TMR
VERSION : 1.0
// stored: InstanceOfName IEC_TIMER
"IEC_TIMER"
BEGIN
END_DATA_BLOCK

DATA_BLOCK "IEC_Timer_0_DB_55"   // DB73
{ S7_Optimized_Access := 'TRUE' }
AUTHOR : Simatic
FAMILY : IEC
NAME : IEC_TMR
VERSION : 1.0
// stored: InstanceOfName IEC_TIMER
"IEC_TIMER"
BEGIN
END_DATA_BLOCK

DATA_BLOCK "IEC_Timer_0_DB_71"   // DB74
{ S7_Optimized_Access := 'TRUE' }
AUTHOR : Simatic
FAMILY : IEC
NAME : IEC_TMR
VERSION : 1.0
// stored: InstanceOfName IEC_TIMER
"IEC_TIMER"
BEGIN
END_DATA_BLOCK

DATA_BLOCK "IEC_Timer_0_DB_72"   // DB75
{ S7_Optimized_Access := 'TRUE' }
AUTHOR : Simatic
FAMILY : IEC
NAME : IEC_TMR
VERSION : 1.0
// stored: InstanceOfName IEC_TIMER
"IEC_TIMER"
BEGIN
END_DATA_BLOCK

DATA_BLOCK "IEC_Timer_0_DB_73"   // DB76
{ S7_Optimized_Access := 'TRUE' }
AUTHOR : Simatic
FAMILY : IEC
NAME : IEC_TMR
VERSION : 1.0
// stored: InstanceOfName IEC_TIMER
"IEC_TIMER"
BEGIN
END_DATA_BLOCK

DATA_BLOCK "IEC_Timer_0_DB_74"   // DB77
{ S7_Optimized_Access := 'TRUE' }
AUTHOR : Simatic
FAMILY : IEC
NAME : IEC_TMR
VERSION : 1.0
// stored: InstanceOfName IEC_TIMER
"IEC_TIMER"
BEGIN
END_DATA_BLOCK

DATA_BLOCK "IEC_Timer_0_DB_75"   // DB78
{ S7_Optimized_Access := 'TRUE' }
AUTHOR : Simatic
FAMILY : IEC
NAME : IEC_TMR
VERSION : 1.0
// stored: InstanceOfName IEC_TIMER
"IEC_TIMER"
BEGIN
END_DATA_BLOCK

DATA_BLOCK "IEC_Timer_0_DB_76"   // DB79
{ S7_Optimized_Access := 'TRUE' }
AUTHOR : Simatic
FAMILY : IEC
NAME : IEC_TMR
VERSION : 1.0
// stored: InstanceOfName IEC_TIMER
"IEC_TIMER"
BEGIN
END_DATA_BLOCK

DATA_BLOCK "IEC_Timer_0_DB_77"   // DB80
{ S7_Optimized_Access := 'TRUE' }
AUTHOR : Simatic
FAMILY : IEC
NAME : IEC_TMR
VERSION : 1.0
// stored: InstanceOfName IEC_TIMER
"IEC_TIMER"
BEGIN
END_DATA_BLOCK

DATA_BLOCK "IEC_Timer_0_DB_78"   // DB81
{ S7_Optimized_Access := 'TRUE' }
AUTHOR : Simatic
FAMILY : IEC
NAME : IEC_TMR
VERSION : 1.0
// stored: InstanceOfName IEC_TIMER
"IEC_TIMER"
BEGIN
END_DATA_BLOCK

DATA_BLOCK "IEC_Timer_0_DB_79"   // DB82
{ S7_Optimized_Access := 'TRUE' }
AUTHOR : Simatic
FAMILY : IEC
NAME : IEC_TMR
VERSION : 1.0
// stored: InstanceOfName IEC_TIMER
"IEC_TIMER"
BEGIN
END_DATA_BLOCK

DATA_BLOCK "IEC_Timer_0_DB_45"   // DB84
{ S7_Optimized_Access := 'TRUE' }
AUTHOR : Simatic
FAMILY : IEC
NAME : IEC_TMR
VERSION : 1.0
// stored: InstanceOfName IEC_TIMER
"IEC_TIMER"
BEGIN
END_DATA_BLOCK

DATA_BLOCK "IEC_Timer_0_DB_56"   // DB85
{ S7_Optimized_Access := 'TRUE' }
AUTHOR : Simatic
FAMILY : IEC
NAME : IEC_TMR
VERSION : 1.0
// stored: InstanceOfName IEC_TIMER
"IEC_TIMER"
BEGIN
END_DATA_BLOCK

DATA_BLOCK "IEC_Timer_0_DB_57"   // DB86
{ S7_Optimized_Access := 'TRUE' }
AUTHOR : Simatic
FAMILY : IEC
NAME : IEC_TMR
VERSION : 1.0
// stored: InstanceOfName IEC_TIMER
"IEC_TIMER"
BEGIN
END_DATA_BLOCK

DATA_BLOCK "IEC_Timer_0_DB_58"   // DB87
{ S7_Optimized_Access := 'TRUE' }
AUTHOR : Simatic
FAMILY : IEC
NAME : IEC_TMR
VERSION : 1.0
// stored: InstanceOfName IEC_TIMER
"IEC_TIMER"
BEGIN
END_DATA_BLOCK

DATA_BLOCK "IEC_Timer_0_DB_59"   // DB88
{ S7_Optimized_Access := 'TRUE' }
AUTHOR : Simatic
FAMILY : IEC
NAME : IEC_TMR
VERSION : 1.0
// stored: InstanceOfName IEC_TIMER
"IEC_TIMER"
BEGIN
END_DATA_BLOCK

DATA_BLOCK "IEC_Timer_0_DB_80"   // DB89
{ S7_Optimized_Access := 'TRUE' }
AUTHOR : Simatic
FAMILY : IEC
NAME : IEC_TMR
VERSION : 1.0
// stored: InstanceOfName IEC_TIMER
"IEC_TIMER"
BEGIN
END_DATA_BLOCK

DATA_BLOCK "IEC_Timer_0_DB_81"   // DB90
{ S7_Optimized_Access := 'TRUE' }
AUTHOR : Simatic
FAMILY : IEC
NAME : IEC_TMR
VERSION : 1.0
// stored: InstanceOfName IEC_TIMER
"IEC_TIMER"
BEGIN
END_DATA_BLOCK

DATA_BLOCK "IEC_Timer_0_DB_82"   // DB91
{ S7_Optimized_Access := 'TRUE' }
AUTHOR : Simatic
FAMILY : IEC
NAME : IEC_TMR
VERSION : 1.0
// stored: InstanceOfName IEC_TIMER
"IEC_TIMER"
BEGIN
END_DATA_BLOCK

DATA_BLOCK "IEC_Timer_0_DB_83"   // DB92
{ S7_Optimized_Access := 'TRUE' }
AUTHOR : Simatic
FAMILY : IEC
NAME : IEC_TMR
VERSION : 1.0
// stored: InstanceOfName IEC_TIMER
"IEC_TIMER"
BEGIN
END_DATA_BLOCK

DATA_BLOCK "IEC_Timer_0_DB_84"   // DB93
{ S7_Optimized_Access := 'TRUE' }
AUTHOR : Simatic
FAMILY : IEC
NAME : IEC_TMR
VERSION : 1.0
// stored: InstanceOfName IEC_TIMER
"IEC_TIMER"
BEGIN
END_DATA_BLOCK

DATA_BLOCK "IEC_Timer_0_DB_85"   // DB94
{ S7_Optimized_Access := 'TRUE' }
AUTHOR : Simatic
FAMILY : IEC
NAME : IEC_TMR
VERSION : 1.0
// stored: InstanceOfName IEC_TIMER
"IEC_TIMER"
BEGIN
END_DATA_BLOCK

DATA_BLOCK "IEC_Timer_0_DB_86"   // DB95
{ S7_Optimized_Access := 'TRUE' }
AUTHOR : Simatic
FAMILY : IEC
NAME : IEC_TMR
VERSION : 1.0
// stored: InstanceOfName IEC_TIMER
"IEC_TIMER"
BEGIN
END_DATA_BLOCK

DATA_BLOCK "IEC_Timer_0_DB_87"   // DB96
{ S7_Optimized_Access := 'TRUE' }
AUTHOR : Simatic
FAMILY : IEC
NAME : IEC_TMR
VERSION : 1.0
// stored: InstanceOfName IEC_TIMER
"IEC_TIMER"
BEGIN
END_DATA_BLOCK

DATA_BLOCK "IEC_Timer_0_DB_88"   // DB97
{ S7_Optimized_Access := 'TRUE' }
AUTHOR : Simatic
FAMILY : IEC
NAME : IEC_TMR
VERSION : 1.0
// stored: InstanceOfName IEC_TIMER
"IEC_TIMER"
BEGIN
END_DATA_BLOCK

DATA_BLOCK "IEC_Timer_0_DB_89"   // DB98
{ S7_Optimized_Access := 'TRUE' }
AUTHOR : Simatic
FAMILY : IEC
NAME : IEC_TMR
VERSION : 1.0
// stored: InstanceOfName IEC_TIMER
"IEC_TIMER"
BEGIN
END_DATA_BLOCK

DATA_BLOCK "IEC_Timer_0_DB_90"   // DB99
{ S7_Optimized_Access := 'TRUE' }
AUTHOR : Simatic
FAMILY : IEC
NAME : IEC_TMR
VERSION : 1.0
// stored: InstanceOfName IEC_TIMER
"IEC_TIMER"
BEGIN
END_DATA_BLOCK

DATA_BLOCK "IEC_Timer_0_DB_91"   // DB100
{ S7_Optimized_Access := 'TRUE' }
AUTHOR : Simatic
FAMILY : IEC
NAME : IEC_TMR
VERSION : 1.0
// stored: InstanceOfName IEC_TIMER
"IEC_TIMER"
BEGIN
END_DATA_BLOCK

DATA_BLOCK "IEC_Timer_0_DB_92"   // DB101
{ S7_Optimized_Access := 'TRUE' }
AUTHOR : Simatic
FAMILY : IEC
NAME : IEC_TMR
VERSION : 1.0
// stored: InstanceOfName IEC_TIMER
"IEC_TIMER"
BEGIN
END_DATA_BLOCK

DATA_BLOCK "IEC_Timer_0_DB_93"   // DB102
{ S7_Optimized_Access := 'TRUE' }
AUTHOR : Simatic
FAMILY : IEC
NAME : IEC_TMR
VERSION : 1.0
// stored: InstanceOfName IEC_TIMER
"IEC_TIMER"
BEGIN
END_DATA_BLOCK

DATA_BLOCK "IEC_Timer_0_DB_94"   // DB103
{ S7_Optimized_Access := 'TRUE' }
AUTHOR : Simatic
FAMILY : IEC
NAME : IEC_TMR
VERSION : 1.0
// stored: InstanceOfName IEC_TIMER
"IEC_TIMER"
BEGIN
END_DATA_BLOCK

DATA_BLOCK "IEC_Timer_0_DB_95"   // DB104
{ S7_Optimized_Access := 'TRUE' }
AUTHOR : Simatic
FAMILY : IEC
NAME : IEC_TMR
VERSION : 1.0
// stored: InstanceOfName IEC_TIMER
"IEC_TIMER"
BEGIN
END_DATA_BLOCK

DATA_BLOCK "IEC_Timer_0_DB_96"   // DB105
{ S7_Optimized_Access := 'TRUE' }
AUTHOR : Simatic
FAMILY : IEC
NAME : IEC_TMR
VERSION : 1.0
// stored: InstanceOfName IEC_TIMER
"IEC_TIMER"
BEGIN
END_DATA_BLOCK

DATA_BLOCK "IEC_Timer_0_DB_97"   // DB106
{ S7_Optimized_Access := 'TRUE' }
AUTHOR : Simatic
FAMILY : IEC
NAME : IEC_TMR
VERSION : 1.0
// stored: InstanceOfName IEC_TIMER
"IEC_TIMER"
BEGIN
END_DATA_BLOCK

DATA_BLOCK "IEC_Timer_0_DB_98"   // DB107
{ S7_Optimized_Access := 'TRUE' }
AUTHOR : Simatic
FAMILY : IEC
NAME : IEC_TMR
VERSION : 1.0
// stored: InstanceOfName IEC_TIMER
"IEC_TIMER"
BEGIN
END_DATA_BLOCK

DATA_BLOCK "IEC_Timer_0_DB_99"   // DB108
{ S7_Optimized_Access := 'TRUE' }
AUTHOR : Simatic
FAMILY : IEC
NAME : IEC_TMR
VERSION : 1.0
// stored: InstanceOfName IEC_TIMER
"IEC_TIMER"
BEGIN
END_DATA_BLOCK

DATA_BLOCK "IEC_Timer_0_DB_100"   // DB109
{ S7_Optimized_Access := 'TRUE' }
AUTHOR : Simatic
FAMILY : IEC
NAME : IEC_TMR
VERSION : 1.0
// stored: InstanceOfName IEC_TIMER
"IEC_TIMER"
BEGIN
END_DATA_BLOCK

DATA_BLOCK "IEC_Timer_0_DB_101"   // DB110
{ S7_Optimized_Access := 'TRUE' }
AUTHOR : Simatic
FAMILY : IEC
NAME : IEC_TMR
VERSION : 1.0
// stored: InstanceOfName IEC_TIMER
"IEC_TIMER"
BEGIN
END_DATA_BLOCK

DATA_BLOCK "IEC_Timer_0_DB_102"   // DB111
{ S7_Optimized_Access := 'TRUE' }
AUTHOR : Simatic
FAMILY : IEC
NAME : IEC_TMR
VERSION : 1.0
// stored: InstanceOfName IEC_TIMER
"IEC_TIMER"
BEGIN
END_DATA_BLOCK

DATA_BLOCK "IEC_Timer_0_DB_103"   // DB112
{ S7_Optimized_Access := 'TRUE' }
AUTHOR : Simatic
FAMILY : IEC
NAME : IEC_TMR
VERSION : 1.0
// stored: InstanceOfName IEC_TIMER
"IEC_TIMER"
BEGIN
END_DATA_BLOCK

DATA_BLOCK "IEC_Timer_0_DB_104"   // DB113
{ S7_Optimized_Access := 'TRUE' }
AUTHOR : Simatic
FAMILY : IEC
NAME : IEC_TMR
VERSION : 1.0
// stored: InstanceOfName IEC_TIMER
"IEC_TIMER"
BEGIN
END_DATA_BLOCK

DATA_BLOCK "IEC_Timer_0_DB_106"   // DB114
{ S7_Optimized_Access := 'TRUE' }
AUTHOR : Simatic
FAMILY : IEC
NAME : IEC_TMR
VERSION : 1.0
// stored: InstanceOfName IEC_TIMER
"IEC_TIMER"
BEGIN
END_DATA_BLOCK

DATA_BLOCK "IEC_Timer_0_DB_107"   // DB115
{ S7_Optimized_Access := 'TRUE' }
AUTHOR : Simatic
FAMILY : IEC
NAME : IEC_TMR
VERSION : 1.0
// stored: InstanceOfName IEC_TIMER
"IEC_TIMER"
BEGIN
END_DATA_BLOCK

// folder: (top level)

FUNCTION_BLOCK "FB_GC_3Lift_10Floor"   // FB1, SCL
{ S7_Optimized_Access := 'TRUE' }
   VAR_INPUT
      HallUpBtn : Array[1..10] of Bool;
      HallDownBtn : Array[1..10] of Bool;
      LiftCarCall : Array[1..3, 1..10] of Bool;
      LiftGroupEnable : Array[1..3] of Bool;
      LiftLocked : Array[1..3] of Bool;
      LiftDisabled : Array[1..3] of Bool;
      LiftFloor : Array[1..3] of Int;
      LiftDir : Array[1..3] of Int;
      LiftRunning : Array[1..3] of Bool;
      LiftDoorOpen : Array[1..3] of Bool;
      LiftLoadPercent : Array[1..3] of Int;
      LiftPower_kW : Array[1..3] of Real;
      GroupMode : Int;
      CycleTime_s : Real;
      LongWaitLimit_s : Real;
      FullLoadLimitPercent : Int;
      EmptyLoadLimitPercent : Int;
      W_Distance : Int;
      W_Direction : Int;
      W_Task : Int;
      W_AheadTask : Int;
      W_LoadPercent : Real;
      empty : Int;
      RideFinishPulse : Array[1..3] of Bool;
      RideTimeSample_s : Array[1..3] of Real;
      HallUpCancel : Array[1..10] of Bool;
      HallDownCancel : Array[1..10] of Bool;
   END_VAR
   VAR_OUTPUT
      AssignedLiftUp : Array[1..10] of Int;
      AssignedLiftDown : Array[1..10] of Int;
      LiftTaskCount : Array[1..3] of Int;
      AheadTaskCountOut : Array[1..3] of Int;
      AvgWait_s : Real;
      CurrentAvgWait_s : Real;
      CurrentWaitingCount : Int;
      LongWaitRatePercent : Real;
      AvgRideTime_s : Real;
      LiftEfficiencyPercent : Array[1..3] of Real;
      SystemEmptyRatePercent : Real;
      LiftEnergy_kWh : Array[1..3] of Real;
      SystemEnergy_kWh : Real;
      HallUpLampOut : Array[1..10] of Bool;
      HallDownLampOut : Array[1..10] of Bool;
   END_VAR
   VAR_IN_OUT
      LiftHallUp : Array[1..3, 1..10] of Bool;
      LiftHallDown : Array[1..3, 1..10] of Bool;
   END_VAR
   VAR
      PrevHallUpBtn : Array[1..10] of Bool;
      PrevHallDownBtn : Array[1..10] of Bool;
      PendingUp : Array[1..10] of Bool;
      PendingDown : Array[1..10] of Bool;
      AssignedUp : Array[1..10] of Int;
      AssignedDown : Array[1..10] of Int;
      WaitUp_s : Array[1..10] of Real;
      WaitDown_s : Array[1..10] of Real;
      LongFlagUp : Array[1..10] of Bool;
      LongFlagDown : Array[1..10] of Bool;
      TotalCallCnt : DInt;
      ServedCallCnt : DInt;
      LongWaitCnt : DInt;
      TotalWait_s : Real;
      TotalRideTime_s : Real;
      RideCnt : DInt;
      PrevRideFinishPulse : Array[1..3] of Bool;
      OnlineTime_s : Array[1..3] of Real;
      RunTime_s : Array[1..3] of Real;
      EmptyRunTime_s : Array[1..3] of Real;
      Energy_kWh : Array[1..3] of Real;
      idxLift : Int;
      idxFloor : Int;
      bestLift : Int;
      bestScore : Int;
      score : Int;
      tmpCycleTime_s : Real;
      tmpLongWaitLimit_s : Real;
      tmpFullLoadLimit : Int;
      tmpEmptyLoadLimit : Int;
      tmpW_Distance : Int;
      tmpW_Direction : Int;
      tmpW_Task : Int;
      tmpW_AheadTask : Int;
      tmpW_LoadPercent : Real;
      ServiceEnable : Array[1..3, 1..10] of Bool;
      canUse : Bool;
      AheadTaskCount : Array[1..3] of Int;
      tmpLiftTaskCount : Array[1..3] of Int;
      curFloor : Int;
      sumRun : Real;
      sumEmptyRun : Real;
      sumActiveWait : Real;
      LastRunDir : Array[1..3] of Int;
      DoorServiceDir : Array[1..3] of Int;
      PrevDoorOpen_GC : Array[1..3] of Bool;
   END_VAR
   VAR_TEMP
      hasUpHere : Bool;
      hasDownHere : Bool;
   END_VAR
BEGIN
   // ================================================================
   // 三部十层电梯群控算法——偶发外呼无法消除完整修正版
   //
   // 本版基于“外部取消优先完整版”修改，解决以下问题：
   // 1. 原程序先执行到站消号、后执行派梯：若电梯已经在该层开门，
   //    呼叫在同一扫描周期或开门保持期间才被派给该梯，会错过消号时机；
   // 2. 原程序优先把 LiftDir / LastRunDir 当作服务方向，电梯在任意楼层
   //    换向时，到站前运行方向可能与实际响应的外呼方向相反；
   // 3. 原程序只在开门上升沿判断服务方向，开门后才完成派梯时不会补判；
   // 4. 同层上下呼若同时被派给同一台梯，无法可靠判断本次开门应消哪一侧。
   //
   // 核心处理：
   // A. 执行顺序改为：采集 -> 统计 -> 派梯 -> 到站消号 -> 灯输出；
   // B. 本层只分配了上呼时，无论到站前运动方向如何，都按上呼服务；
   // C. 本层只分配了下呼时，无论到站前运动方向如何，都按下呼服务；
   // D. 门已经打开但服务方向仍为 0 时，允许根据后来完成的派梯结果补判；
   // E. 禁止同层相反方向外呼同时派给同一台梯；若检测到旧状态冲突，
   //    先回收上下呼并重新派梯；
   // F. 一次开门过程中 DoorServiceDir 锁存，避免先后把上下呼都消除；
   // G. 外呼灯仍由群控唯一输出，外部程序通过 HallUpCancel / HallDownCancel
   //    取消内部任务，不要直接与群控同时写 HallUpLampOut / HallDownLampOut。
   //
   // VAR_INPUT 中新增/保留：
   //     HallUpCancel   : ARRAY[1..10] OF BOOL;
   //     HallDownCancel : ARRAY[1..10] OF BOOL;
   //
   // VAR_OUTPUT 中新增/保留：
   //     HallUpLampOut   : ARRAY[1..10] OF BOOL;
   //     HallDownLampOut : ARRAY[1..10] OF BOOL;
   //
   // FB Static（VAR）中新增/保留：
   //     LastRunDir      : ARRAY[1..3] OF INT;
   //     DoorServiceDir  : ARRAY[1..3] OF INT;
   //     PrevDoorOpen_GC : ARRAY[1..3] OF BOOL;
   //
   // VAR_TEMP 中新增：
   //     hasUpHere   : BOOL;
   //     hasDownHere : BOOL;
   //
   // 方向定义：1=上行服务，-1=下行服务，0=未确定。
   // ================================================================

   // ==================================================
   // 0. 参数默认值保护
   // ==================================================
   IF #CycleTime_s <= 0.0 THEN
       #tmpCycleTime_s := 0.1;
   ELSE
       #tmpCycleTime_s := #CycleTime_s;
   END_IF;

   IF #LongWaitLimit_s <= 0.0 THEN
       #tmpLongWaitLimit_s := 60.0;
   ELSE
       #tmpLongWaitLimit_s := #LongWaitLimit_s;
   END_IF;

   IF #FullLoadLimitPercent <= 0 THEN
       #tmpFullLoadLimit := 95;
   ELSE
       #tmpFullLoadLimit := #FullLoadLimitPercent;
   END_IF;

   IF #EmptyLoadLimitPercent < 0 THEN
       #tmpEmptyLoadLimit := 5;
   ELSE
       #tmpEmptyLoadLimit := #EmptyLoadLimitPercent;
   END_IF;

   IF #W_Distance <= 0 THEN
       #tmpW_Distance := 10;
   ELSE
       #tmpW_Distance := #W_Distance;
   END_IF;

   IF #W_Direction <= 0 THEN
       #tmpW_Direction := 30;
   ELSE
       #tmpW_Direction := #W_Direction;
   END_IF;

   IF #W_Task <= 0 THEN
       #tmpW_Task := 6;
   ELSE
       #tmpW_Task := #W_Task;
   END_IF;

   IF #W_AheadTask <= 0 THEN
       #tmpW_AheadTask := 8;
   ELSE
       #tmpW_AheadTask := #W_AheadTask;
   END_IF;

   IF #W_LoadPercent <= 0.0 THEN
       #tmpW_LoadPercent := 0.2;
   ELSE
       #tmpW_LoadPercent := #W_LoadPercent;
   END_IF;

   // ==================================================
   // 1. 动态分区服务表
   // ==================================================
   FOR #idxLift := 1 TO 3 DO
       FOR #idxFloor := 1 TO 10 DO

           IF #GroupMode = 0 THEN
               #ServiceEnable[#idxLift, #idxFloor] := TRUE;

           ELSIF #GroupMode = 1 THEN
               IF #idxLift = 1 THEN
                   #ServiceEnable[#idxLift, #idxFloor] := (#idxFloor >= 1) AND (#idxFloor <= 5);
               ELSIF #idxLift = 2 THEN
                   #ServiceEnable[#idxLift, #idxFloor] := (#idxFloor = 1) OR (#idxFloor >= 6);
               ELSE
                   #ServiceEnable[#idxLift, #idxFloor] := TRUE;
               END_IF;

           ELSIF #GroupMode = 2 THEN
               IF #idxLift = 1 THEN
                   #ServiceEnable[#idxLift, #idxFloor] := (#idxFloor >= 1) AND (#idxFloor <= 5);
               ELSIF #idxLift = 2 THEN
                   #ServiceEnable[#idxLift, #idxFloor] := (#idxFloor >= 6) AND (#idxFloor <= 10);
               ELSE
                   #ServiceEnable[#idxLift, #idxFloor] := TRUE;
               END_IF;

           ELSIF #GroupMode = 3 THEN
               IF #idxLift = 1 THEN
                   #ServiceEnable[#idxLift, #idxFloor] := (#idxFloor >= 1) AND (#idxFloor <= 6);
               ELSIF #idxLift = 2 THEN
                   #ServiceEnable[#idxLift, #idxFloor] := (#idxFloor >= 5) AND (#idxFloor <= 10);
               ELSE
                   #ServiceEnable[#idxLift, #idxFloor] := TRUE;
               END_IF;

           ELSIF #GroupMode = 4 THEN
               IF #idxLift = 1 THEN
                   #ServiceEnable[#idxLift, #idxFloor] := (#idxFloor >= 1) AND (#idxFloor <= 4);
               ELSIF #idxLift = 2 THEN
                   #ServiceEnable[#idxLift, #idxFloor] := (#idxFloor >= 4) AND (#idxFloor <= 7);
               ELSE
                   #ServiceEnable[#idxLift, #idxFloor] := (#idxFloor >= 7) AND (#idxFloor <= 10);
               END_IF;

           ELSE
               #ServiceEnable[#idxLift, #idxFloor] := TRUE;
           END_IF;

       END_FOR;
   END_FOR;

   // ==================================================
   // 2. 无效楼层清除
   // ==================================================
   FOR #idxLift := 1 TO 3 DO
       #LiftHallUp[#idxLift, 10] := FALSE;
       #LiftHallDown[#idxLift, 1] := FALSE;
   END_FOR;

   // ==================================================
   // 3. 锁梯 / 禁用 / 退出群控 / 分区变化时回收任务
   // ==================================================
   FOR #idxFloor := 1 TO 9 DO
       #idxLift := #AssignedUp[#idxFloor];

       IF (#idxLift >= 1) AND (#idxLift <= 3) THEN
           IF (NOT #LiftGroupEnable[#idxLift]) OR #LiftLocked[#idxLift] OR #LiftDisabled[#idxLift] OR
               (NOT #ServiceEnable[#idxLift, #idxFloor]) THEN

               #PendingUp[#idxFloor] := TRUE;
               #AssignedUp[#idxFloor] := 0;
               #LiftHallUp[#idxLift, #idxFloor] := FALSE;
           END_IF;
       ELSE
           #AssignedUp[#idxFloor] := 0;
       END_IF;
   END_FOR;

   FOR #idxFloor := 2 TO 10 DO
       #idxLift := #AssignedDown[#idxFloor];

       IF (#idxLift >= 1) AND (#idxLift <= 3) THEN
           IF (NOT #LiftGroupEnable[#idxLift]) OR #LiftLocked[#idxLift] OR #LiftDisabled[#idxLift] OR
               (NOT #ServiceEnable[#idxLift, #idxFloor]) THEN

               #PendingDown[#idxFloor] := TRUE;
               #AssignedDown[#idxFloor] := 0;
               #LiftHallDown[#idxLift, #idxFloor] := FALSE;
           END_IF;
       ELSE
           #AssignedDown[#idxFloor] := 0;
       END_IF;
   END_FOR;

   FOR #idxLift := 1 TO 3 DO
       IF (NOT #LiftGroupEnable[#idxLift]) OR #LiftLocked[#idxLift] OR #LiftDisabled[#idxLift] THEN
           FOR #idxFloor := 1 TO 10 DO
               #LiftHallUp[#idxLift, #idxFloor] := FALSE;
               #LiftHallDown[#idxLift, #idxFloor] := FALSE;
           END_FOR;
       END_IF;
   END_FOR;

   // ==================================================
   // 4. 外部取消优先处理及外呼按钮上升沿采集
   // ==================================================
   // 重要：
   // 1. 外部自动程序不要直接写 HallUpLampOut / HallDownLampOut；
   // 2. 需要自动复位某层外呼时，应给 HallUpCancel / HallDownCancel；
   // 3. 群控收到取消命令后，必须同时清除内部任务状态，指示灯才不会被重新置位。

   // --------------------------------------------------
   // 4.1 上呼：取消优先，未取消时才采集上升沿
   // --------------------------------------------------
   FOR #idxFloor := 1 TO 9 DO

       // 外部取消命令优先级最高。
       IF #HallUpCancel[#idxFloor] THEN

           // 清除三台电梯在该层可能残留的上呼任务位。
           // 即使 AssignedUp 异常或已经被其他逻辑清零，也能彻底清除残留任务。
           FOR #idxLift := 1 TO 3 DO
               #LiftHallUp[#idxLift, #idxFloor] := FALSE;
           END_FOR;

           // 清除群控内部的待分配和已分配状态。
           #PendingUp[#idxFloor] := FALSE;
           #AssignedUp[#idxFloor] := 0;

           // 清除本次仍在活动的等待状态。
           #WaitUp_s[#idxFloor] := 0.0;
           #LongFlagUp[#idxFloor] := FALSE;

           // 把当前按钮状态写入沿记忆。
           // 如果按钮仍为 TRUE，取消解除后不会立即被当成新的上升沿。
           #PrevHallUpBtn[#idxFloor] := #HallUpBtn[#idxFloor];

           // 没有取消命令时，才允许正常登记新的上呼。
       ELSIF #HallUpBtn[#idxFloor] AND (NOT #PrevHallUpBtn[#idxFloor]) THEN

           IF (NOT #PendingUp[#idxFloor]) AND (#AssignedUp[#idxFloor] = 0) THEN
               #PendingUp[#idxFloor] := TRUE;
               #WaitUp_s[#idxFloor] := 0.0;
               #LongFlagUp[#idxFloor] := FALSE;
               #TotalCallCnt := #TotalCallCnt + 1;
           END_IF;
       END_IF;

       // 正常保存按钮当前状态。
       // 取消分支中虽然已经写过一次，再写相同值不会产生副作用。
       #PrevHallUpBtn[#idxFloor] := #HallUpBtn[#idxFloor];
   END_FOR;


   // --------------------------------------------------
   // 4.2 下呼：取消优先，未取消时才采集上升沿
   // --------------------------------------------------
   FOR #idxFloor := 2 TO 10 DO

       // 外部取消命令优先级最高。
       IF #HallDownCancel[#idxFloor] THEN

           // 清除三台电梯在该层可能残留的下呼任务位。
           FOR #idxLift := 1 TO 3 DO
               #LiftHallDown[#idxLift, #idxFloor] := FALSE;
           END_FOR;

           // 清除群控内部的待分配和已分配状态。
           #PendingDown[#idxFloor] := FALSE;
           #AssignedDown[#idxFloor] := 0;

           // 清除本次仍在活动的等待状态。
           #WaitDown_s[#idxFloor] := 0.0;
           #LongFlagDown[#idxFloor] := FALSE;

           // 同步按钮沿记忆，避免取消解除后按钮仍为 TRUE 而立即重新登记。
           #PrevHallDownBtn[#idxFloor] := #HallDownBtn[#idxFloor];

           // 没有取消命令时，才允许正常登记新的下呼。
       ELSIF #HallDownBtn[#idxFloor] AND (NOT #PrevHallDownBtn[#idxFloor]) THEN

           IF (NOT #PendingDown[#idxFloor]) AND (#AssignedDown[#idxFloor] = 0) THEN
               #PendingDown[#idxFloor] := TRUE;
               #WaitDown_s[#idxFloor] := 0.0;
               #LongFlagDown[#idxFloor] := FALSE;
               #TotalCallCnt := #TotalCallCnt + 1;
           END_IF;
       END_IF;

       // 正常保存按钮当前状态。
       #PrevHallDownBtn[#idxFloor] := #HallDownBtn[#idxFloor];
   END_FOR;

   // ==================================================
   // 5. 清理同层上下呼被分配给同一台梯的冲突状态
   // ==================================================
   // 同一层的上呼和下呼不能同时由同一台梯持有，否则在换向层无法仅凭
   // 到站前运动方向确定本次开门究竟服务哪一侧。
   // 检测到旧状态冲突时，两侧都回收到 Pending，随后由本扫描周期的
   // 派梯段重新分配；新的派梯逻辑也会禁止再次派给同一台梯。
   FOR #idxFloor := 2 TO 9 DO
       IF (#AssignedUp[#idxFloor] >= 1)
           AND (#AssignedUp[#idxFloor] <= 3)
           AND (#AssignedUp[#idxFloor] = #AssignedDown[#idxFloor]) THEN

           #idxLift := #AssignedUp[#idxFloor];

           #LiftHallUp[#idxLift, #idxFloor] := FALSE;
           #LiftHallDown[#idxLift, #idxFloor] := FALSE;

           // 若冲突发生时该梯正在本层开门，清除旧的服务方向锁存，
           // 让后面的重新派梯结果能够在同一扫描周期重新判断。
           IF (#LiftFloor[#idxLift] = #idxFloor) AND #LiftDoorOpen[#idxLift] THEN
               #DoorServiceDir[#idxLift] := 0;
           END_IF;

           #AssignedUp[#idxFloor] := 0;
           #AssignedDown[#idxFloor] := 0;

           IF NOT #HallUpCancel[#idxFloor] THEN
               #PendingUp[#idxFloor] := TRUE;
           ELSE
               #PendingUp[#idxFloor] := FALSE;
           END_IF;

           IF NOT #HallDownCancel[#idxFloor] THEN
               #PendingDown[#idxFloor] := TRUE;
           ELSE
               #PendingDown[#idxFloor] := FALSE;
           END_IF;
       END_IF;
   END_FOR;


   // ==================================================
   // 6. 派梯前统计每部电梯总任务数量
   // ==================================================
   FOR #idxLift := 1 TO 3 DO
       #tmpLiftTaskCount[#idxLift] := 0;
   END_FOR;

   FOR #idxLift := 1 TO 3 DO

       FOR #idxFloor := 1 TO 9 DO
           IF #LiftHallUp[#idxLift, #idxFloor] THEN
               #tmpLiftTaskCount[#idxLift] := #tmpLiftTaskCount[#idxLift] + 1;
           END_IF;
       END_FOR;

       FOR #idxFloor := 2 TO 10 DO
           IF #LiftHallDown[#idxLift, #idxFloor] THEN
               #tmpLiftTaskCount[#idxLift] := #tmpLiftTaskCount[#idxLift] + 1;
           END_IF;
       END_FOR;

       FOR #idxFloor := 1 TO 10 DO
           IF #LiftCarCall[#idxLift, #idxFloor] THEN
               #tmpLiftTaskCount[#idxLift] := #tmpLiftTaskCount[#idxLift] + 1;
           END_IF;
       END_FOR;

   END_FOR;

   // ==================================================
   // 7. 统计前方任务数量
   // ==================================================
   FOR #idxLift := 1 TO 3 DO
       #AheadTaskCount[#idxLift] := 0;

       #curFloor := #LiftFloor[#idxLift];

       IF #curFloor < 1 THEN
           #curFloor := 1;
       ELSIF #curFloor > 10 THEN
           #curFloor := 10;
       END_IF;

       IF #LiftDir[#idxLift] = 1 THEN

           IF #curFloor < 10 THEN
               FOR #idxFloor := #curFloor + 1 TO 10 DO

                   IF #LiftCarCall[#idxLift, #idxFloor] THEN
                       #AheadTaskCount[#idxLift] := #AheadTaskCount[#idxLift] + 1;
                   END_IF;

                   IF #idxFloor <= 9 THEN
                       IF #LiftHallUp[#idxLift, #idxFloor] THEN
                           #AheadTaskCount[#idxLift] := #AheadTaskCount[#idxLift] + 1;
                       END_IF;
                   END_IF;

                   IF #idxFloor >= 2 THEN
                       IF #LiftHallDown[#idxLift, #idxFloor] THEN
                           #AheadTaskCount[#idxLift] := #AheadTaskCount[#idxLift] + 1;
                       END_IF;
                   END_IF;

               END_FOR;
           END_IF;

       ELSIF #LiftDir[#idxLift] = -1 THEN

           IF #curFloor > 1 THEN
               FOR #idxFloor := 1 TO #curFloor - 1 DO

                   IF #LiftCarCall[#idxLift, #idxFloor] THEN
                       #AheadTaskCount[#idxLift] := #AheadTaskCount[#idxLift] + 1;
                   END_IF;

                   IF #idxFloor <= 9 THEN
                       IF #LiftHallUp[#idxLift, #idxFloor] THEN
                           #AheadTaskCount[#idxLift] := #AheadTaskCount[#idxLift] + 1;
                       END_IF;
                   END_IF;

                   IF #idxFloor >= 2 THEN
                       IF #LiftHallDown[#idxLift, #idxFloor] THEN
                           #AheadTaskCount[#idxLift] := #AheadTaskCount[#idxLift] + 1;
                       END_IF;
                   END_IF;

               END_FOR;
           END_IF;

       ELSE
           #AheadTaskCount[#idxLift] := 0;
       END_IF;

       #AheadTaskCountOut[#idxLift] := #AheadTaskCount[#idxLift];

   END_FOR;

   // ==================================================
   // 8. 分配上呼、下呼请求
   // ==================================================
   // 新增限制：中间楼层相反方向的呼叫如果已经分配给某台电梯，另一方向
   // 不再分配给同一台梯。只有其他电梯可用时才分给其他梯；如果只有一台
   // 梯可用，则另一方向继续 Pending，等第一方向完成后再重新分配。

   // --------------------------------------------------
   // 8.1 分配上呼请求
   // --------------------------------------------------
   FOR #idxFloor := 1 TO 9 DO
       IF #PendingUp[#idxFloor] AND (NOT #HallUpCancel[#idxFloor]) THEN
           #bestLift := 0;
           #bestScore := 32000;

           FOR #idxLift := 1 TO 3 DO
               #canUse :=
               #LiftGroupEnable[#idxLift] AND
               (NOT #LiftLocked[#idxLift]) AND
               (NOT #LiftDisabled[#idxLift]) AND
               #ServiceEnable[#idxLift, #idxFloor] AND
               (#LiftLoadPercent[#idxLift] < #tmpFullLoadLimit) AND
               // 2～9层若下呼已派给本梯，上呼不得再派给同一台梯。
               ((#idxFloor = 1) OR (#AssignedDown[#idxFloor] <> #idxLift));

               #score := "FC_GC_Score"(
                                       ReqFloor := #idxFloor,
                                       ReqDir := 1,
                                       LiftFloor := #LiftFloor[#idxLift],
                                       LiftDir := #LiftDir[#idxLift],
                                       LiftRunning := #LiftRunning[#idxLift],
                                       LiftLoadPercent := #LiftLoadPercent[#idxLift],
                                       TaskCount := #tmpLiftTaskCount[#idxLift],
                                       AheadTaskCount := #AheadTaskCount[#idxLift],
                                       CanUse := #canUse,
                                       W_Distance := #tmpW_Distance,
                                       W_Direction := #tmpW_Direction,
                                       W_Task := #tmpW_Task,
                                       W_AheadTask := #tmpW_AheadTask,
                                       W_LoadPercent := #tmpW_LoadPercent,
                                       empty := #empty
               );

               IF #score < #bestScore THEN
                   #bestScore := #score;
                   #bestLift := #idxLift;
               END_IF;
           END_FOR;

           IF #bestLift <> 0 THEN
               #LiftHallUp[#bestLift, #idxFloor] := TRUE;
               #AssignedUp[#idxFloor] := #bestLift;
               #PendingUp[#idxFloor] := FALSE;
               #tmpLiftTaskCount[#bestLift] := #tmpLiftTaskCount[#bestLift] + 1;
           END_IF;
       END_IF;
   END_FOR;


   // --------------------------------------------------
   // 8.2 分配下呼请求
   // --------------------------------------------------
   FOR #idxFloor := 2 TO 10 DO
       IF #PendingDown[#idxFloor] AND (NOT #HallDownCancel[#idxFloor]) THEN
           #bestLift := 0;
           #bestScore := 32000;

           FOR #idxLift := 1 TO 3 DO
               #canUse :=
               #LiftGroupEnable[#idxLift] AND
               (NOT #LiftLocked[#idxLift]) AND
               (NOT #LiftDisabled[#idxLift]) AND
               #ServiceEnable[#idxLift, #idxFloor] AND
               (#LiftLoadPercent[#idxLift] < #tmpFullLoadLimit) AND
               // 2～9层若上呼已派给本梯，下呼不得再派给同一台梯。
               ((#idxFloor = 10) OR (#AssignedUp[#idxFloor] <> #idxLift));

               #score := "FC_GC_Score"(
                                       ReqFloor := #idxFloor,
                                       ReqDir := -1,
                                       LiftFloor := #LiftFloor[#idxLift],
                                       LiftDir := #LiftDir[#idxLift],
                                       LiftRunning := #LiftRunning[#idxLift],
                                       LiftLoadPercent := #LiftLoadPercent[#idxLift],
                                       TaskCount := #tmpLiftTaskCount[#idxLift],
                                       AheadTaskCount := #AheadTaskCount[#idxLift],
                                       CanUse := #canUse,
                                       W_Distance := #tmpW_Distance,
                                       W_Direction := #tmpW_Direction,
                                       W_Task := #tmpW_Task,
                                       W_AheadTask := #tmpW_AheadTask,
                                       W_LoadPercent := #tmpW_LoadPercent,
                                       empty := #empty
               );

               IF #score < #bestScore THEN
                   #bestScore := #score;
                   #bestLift := #idxLift;
               END_IF;
           END_FOR;

           IF #bestLift <> 0 THEN
               #LiftHallDown[#bestLift, #idxFloor] := TRUE;
               #AssignedDown[#idxFloor] := #bestLift;
               #PendingDown[#idxFloor] := FALSE;
               #tmpLiftTaskCount[#bestLift] := #tmpLiftTaskCount[#bestLift] + 1;
           END_IF;
       END_IF;
   END_FOR;


   // ==================================================
   // 9. 派梯完成后判断开门服务方向，并消除对应外呼
   // ==================================================
   // 关键原则：
   // 1. 本层只有上呼分配给本梯：直接认定本次服务上呼，不看到站前方向；
   // 2. 本层只有下呼分配给本梯：直接认定本次服务下呼，不看到站前方向；
   // 3. 本层上下呼同时属于本梯原则上已被第5、8段阻止；若异常仍出现，
   //    才使用 LiftDir / LastRunDir 作为兜底；
   // 4. 判断放在派梯之后，因此电梯已开门后才完成派梯也能在本扫描周期补判；
   // 5. DoorServiceDir 在一次开门过程中锁存，防止相反方向呼叫后来出现时
   //    被同一次开门继续消除。
   FOR #idxLift := 1 TO 3 DO

       // 持续记录最后一个有效物理运行方向，仅用于双向冲突兜底。
       IF (#LiftDir[#idxLift] = 1) OR (#LiftDir[#idxLift] = -1) THEN
           #LastRunDir[#idxLift] := #LiftDir[#idxLift];
       END_IF;

       #curFloor := #LiftFloor[#idxLift];
       IF #curFloor < 1 THEN
           #curFloor := 1;
       ELSIF #curFloor > 10 THEN
           #curFloor := 10;
       END_IF;

       // 本层是否有对应方向的全局外呼实际分配给本梯。
       // 以 Assigned 为消灯状态源，不要求 LiftHall 位仍为 TRUE；这样即使单梯
       // 程序先复位了任务位，只要群控分配记录仍存在，到站时仍可完成消号。
       #hasUpHere := FALSE;
       #hasDownHere := FALSE;

       IF #curFloor <= 9 THEN
           #hasUpHere := (#AssignedUp[#curFloor] = #idxLift);
       END_IF;

       IF #curFloor >= 2 THEN
           #hasDownHere := (#AssignedDown[#curFloor] = #idxLift);
       END_IF;

       IF #LiftDoorOpen[#idxLift] THEN

           // 开门上升沿，或门已打开但之前没有确定服务方向时，允许判断/补判。
           IF (NOT #PrevDoorOpen_GC[#idxLift]) OR (#DoorServiceDir[#idxLift] = 0) THEN

               IF #hasUpHere AND (NOT #hasDownHere) THEN
                   #DoorServiceDir[#idxLift] := 1;

               ELSIF #hasDownHere AND (NOT #hasUpHere) THEN
                   #DoorServiceDir[#idxLift] := -1;

               ELSIF #hasUpHere AND #hasDownHere THEN
                   // 异常双向冲突兜底。正常情况下第5、8段已避免该状态。
                   IF (#LiftDir[#idxLift] = 1) OR (#LiftDir[#idxLift] = -1) THEN
                       #DoorServiceDir[#idxLift] := #LiftDir[#idxLift];
                   ELSIF (#LastRunDir[#idxLift] = 1) OR (#LastRunDir[#idxLift] = -1) THEN
                       #DoorServiceDir[#idxLift] := #LastRunDir[#idxLift];
                   ELSE
                       #DoorServiceDir[#idxLift] := 0;
                   END_IF;

               ELSE
                   // 本层尚无群控外呼分配，不依据旧运行方向预先锁定服务方向。
                   // 如果门保持打开期间呼叫随后派到本梯，下一扫描周期仍可补判。
                   #DoorServiceDir[#idxLift] := 0;
               END_IF;
           END_IF;

           // --------------------------------------------------
           // 9.1 本次开门服务上呼
           // --------------------------------------------------
           IF (#DoorServiceDir[#idxLift] = 1) AND #hasUpHere THEN
               #LiftHallUp[#idxLift, #curFloor] := FALSE;
               #PendingUp[#curFloor] := FALSE;
               #AssignedUp[#curFloor] := 0;

               #ServedCallCnt := #ServedCallCnt + 1;
               #TotalWait_s := #TotalWait_s + #WaitUp_s[#curFloor];
               #WaitUp_s[#curFloor] := 0.0;
               #LongFlagUp[#curFloor] := FALSE;
           END_IF;

           // --------------------------------------------------
           // 9.2 本次开门服务下呼
           // --------------------------------------------------
           IF (#DoorServiceDir[#idxLift] = -1) AND #hasDownHere THEN
               #LiftHallDown[#idxLift, #curFloor] := FALSE;
               #PendingDown[#curFloor] := FALSE;
               #AssignedDown[#curFloor] := 0;

               #ServedCallCnt := #ServedCallCnt + 1;
               #TotalWait_s := #TotalWait_s + #WaitDown_s[#curFloor];
               #WaitDown_s[#curFloor] := 0.0;
               #LongFlagDown[#curFloor] := FALSE;
           END_IF;

       ELSE
           // 门关闭后才允许下一次开门重新确定服务方向。
           #DoorServiceDir[#idxLift] := 0;
       END_IF;

       // 必须在本扫描周期所有开门判断完成后更新沿记忆。
       #PrevDoorOpen_GC[#idxLift] := #LiftDoorOpen[#idxLift];
   END_FOR;


   // ==================================================
   // 10. 等待时间统计
   // ==================================================
   #CurrentWaitingCount := 0;
   #sumActiveWait := 0.0;

   FOR #idxFloor := 1 TO 9 DO
       IF #PendingUp[#idxFloor] OR (#AssignedUp[#idxFloor] <> 0) THEN
           #WaitUp_s[#idxFloor] := #WaitUp_s[#idxFloor] + #tmpCycleTime_s;
           #CurrentWaitingCount := #CurrentWaitingCount + 1;
           #sumActiveWait := #sumActiveWait + #WaitUp_s[#idxFloor];

           IF (#WaitUp_s[#idxFloor] >= #tmpLongWaitLimit_s) AND (NOT #LongFlagUp[#idxFloor]) THEN
               #LongFlagUp[#idxFloor] := TRUE;
               #LongWaitCnt := #LongWaitCnt + 1;
           END_IF;
       END_IF;
   END_FOR;

   FOR #idxFloor := 2 TO 10 DO
       IF #PendingDown[#idxFloor] OR (#AssignedDown[#idxFloor] <> 0) THEN
           #WaitDown_s[#idxFloor] := #WaitDown_s[#idxFloor] + #tmpCycleTime_s;
           #CurrentWaitingCount := #CurrentWaitingCount + 1;
           #sumActiveWait := #sumActiveWait + #WaitDown_s[#idxFloor];

           IF (#WaitDown_s[#idxFloor] >= #tmpLongWaitLimit_s) AND (NOT #LongFlagDown[#idxFloor]) THEN
               #LongFlagDown[#idxFloor] := TRUE;
               #LongWaitCnt := #LongWaitCnt + 1;
           END_IF;
       END_IF;
   END_FOR;

   IF #CurrentWaitingCount > 0 THEN
       #CurrentAvgWait_s := #sumActiveWait / INT_TO_REAL(#CurrentWaitingCount);
   ELSE
       #CurrentAvgWait_s := 0.0;
   END_IF;

   // ==================================================
   // 11. 消号后重新统计每部电梯当前任务数量
   // ==================================================
   // 派梯阶段为了评分已统计过一次；本段在到站消号后重新统计，确保
   // LiftTaskCount 输出不会在快速“派梯并立即消号”场景中多保留一个扫描周期。
   FOR #idxLift := 1 TO 3 DO
       #tmpLiftTaskCount[#idxLift] := 0;

       FOR #idxFloor := 1 TO 9 DO
           IF #LiftHallUp[#idxLift, #idxFloor] THEN
               #tmpLiftTaskCount[#idxLift] := #tmpLiftTaskCount[#idxLift] + 1;
           END_IF;
       END_FOR;

       FOR #idxFloor := 2 TO 10 DO
           IF #LiftHallDown[#idxLift, #idxFloor] THEN
               #tmpLiftTaskCount[#idxLift] := #tmpLiftTaskCount[#idxLift] + 1;
           END_IF;
       END_FOR;

       FOR #idxFloor := 1 TO 10 DO
           IF #LiftCarCall[#idxLift, #idxFloor] THEN
               #tmpLiftTaskCount[#idxLift] := #tmpLiftTaskCount[#idxLift] + 1;
           END_IF;
       END_FOR;
   END_FOR;


   // ==================================================
   // 12. 输出分配结果及外呼指示灯
   // ==================================================

   // 输出每层上呼、下呼当前分配到的电梯编号
   FOR #idxFloor := 1 TO 10 DO
       #AssignedLiftUp[#idxFloor] := #AssignedUp[#idxFloor];
       #AssignedLiftDown[#idxFloor] := #AssignedDown[#idxFloor];

       // 先清零，随后只对有效楼层重新赋值
       #HallUpLampOut[#idxFloor] := FALSE;
       #HallDownLampOut[#idxFloor] := FALSE;
   END_FOR;

   // 1～9 层有上呼按钮。
   // 请求处于待分配状态，或已经分配给某台电梯时，上呼灯保持点亮。
   // HallUpCancel 为 TRUE 时，无论内部状态如何，当前扫描周期都强制熄灭。
   FOR #idxFloor := 1 TO 9 DO
       #HallUpLampOut[#idxFloor] :=
       (#PendingUp[#idxFloor] OR (#AssignedUp[#idxFloor] <> 0))
       AND (NOT #HallUpCancel[#idxFloor]);
   END_FOR;

   // 2～10 层有下呼按钮。
   // 请求处于待分配状态，或已经分配给某台电梯时，下呼灯保持点亮。
   // HallDownCancel 为 TRUE 时，无论内部状态如何，当前扫描周期都强制熄灭。
   FOR #idxFloor := 2 TO 10 DO
       #HallDownLampOut[#idxFloor] :=
       (#PendingDown[#idxFloor] OR (#AssignedDown[#idxFloor] <> 0))
       AND (NOT #HallDownCancel[#idxFloor]);
   END_FOR;

   // 输出每台电梯当前任务数量
   FOR #idxLift := 1 TO 3 DO
       #LiftTaskCount[#idxLift] := #tmpLiftTaskCount[#idxLift];
   END_FOR;

   // ==================================================
   // 13. 效能统计
   // ==================================================
   #sumRun := 0.0;
   #sumEmptyRun := 0.0;
   #SystemEnergy_kWh := 0.0;

   FOR #idxLift := 1 TO 3 DO

       IF #LiftGroupEnable[#idxLift] AND (NOT #LiftLocked[#idxLift]) AND (NOT #LiftDisabled[#idxLift]) THEN

           #OnlineTime_s[#idxLift] := #OnlineTime_s[#idxLift] + #tmpCycleTime_s;

           IF #LiftRunning[#idxLift] THEN
               #RunTime_s[#idxLift] := #RunTime_s[#idxLift] + #tmpCycleTime_s;

               IF #LiftLoadPercent[#idxLift] <= #tmpEmptyLoadLimit THEN
                   #EmptyRunTime_s[#idxLift] := #EmptyRunTime_s[#idxLift] + #tmpCycleTime_s;
               END_IF;
           END_IF;

           #Energy_kWh[#idxLift] := #Energy_kWh[#idxLift] + (#LiftPower_kW[#idxLift] * #tmpCycleTime_s / 3600.0);
       END_IF;

       IF #OnlineTime_s[#idxLift] > 0.0 THEN
           #LiftEfficiencyPercent[#idxLift] := #RunTime_s[#idxLift] / #OnlineTime_s[#idxLift] * 100.0;
       ELSE
           #LiftEfficiencyPercent[#idxLift] := 0.0;
       END_IF;

       #LiftEnergy_kWh[#idxLift] := #Energy_kWh[#idxLift];

       #sumRun := #sumRun + #RunTime_s[#idxLift];
       #sumEmptyRun := #sumEmptyRun + #EmptyRunTime_s[#idxLift];
       #SystemEnergy_kWh := #SystemEnergy_kWh + #Energy_kWh[#idxLift];

       IF #RideFinishPulse[#idxLift] AND (NOT #PrevRideFinishPulse[#idxLift]) THEN
           IF #RideTimeSample_s[#idxLift] > 0.0 THEN
               #TotalRideTime_s := #TotalRideTime_s + #RideTimeSample_s[#idxLift];
               #RideCnt := #RideCnt + 1;
           END_IF;
       END_IF;

       #PrevRideFinishPulse[#idxLift] := #RideFinishPulse[#idxLift];
   END_FOR;

   IF #sumRun > 0.0 THEN
       #SystemEmptyRatePercent := #sumEmptyRun / #sumRun * 100.0;
   ELSE
       #SystemEmptyRatePercent := 0.0;
   END_IF;

   IF #ServedCallCnt > 0 THEN
       #AvgWait_s := #TotalWait_s / DINT_TO_REAL(#ServedCallCnt);
   ELSE
       #AvgWait_s := 0.0;
   END_IF;

   IF #TotalCallCnt > 0 THEN
       #LongWaitRatePercent := DINT_TO_REAL(#LongWaitCnt) / DINT_TO_REAL(#TotalCallCnt) * 100.0;
   ELSE
       #LongWaitRatePercent := 0.0;
   END_IF;

   IF #RideCnt > 0 THEN
       #AvgRideTime_s := #TotalRideTime_s / DINT_TO_REAL(#RideCnt);
   ELSE
       #AvgRideTime_s := 0.0;
   END_IF;
END_FUNCTION_BLOCK

FUNCTION "外呼分配" : Void   // FC1, LAD
{ S7_Optimized_Access := 'TRUE' }
VERSION : 0.1
   VAR_TEMP   // added for the SCL form of the ladder/FBD networks
      _w1 : Bool;
      _w2 : Bool;
      _w3 : Bool;
      _w4 : Bool;
      _w5 : Bool;
      _w6 : Bool;
      _w7 : Bool;
      _w8 : Bool;
      _w9 : Bool;
      _w10 : Bool;
      _w11 : Bool;
      _w12 : Bool;
      _w13 : Bool;
      _w14 : Bool;
      _w15 : Bool;
      _w16 : Bool;
      _w17 : Bool;
      _w18 : Bool;
   END_VAR
BEGIN

REGION Network 1: 外呼上下行按钮指示灯及上下呼
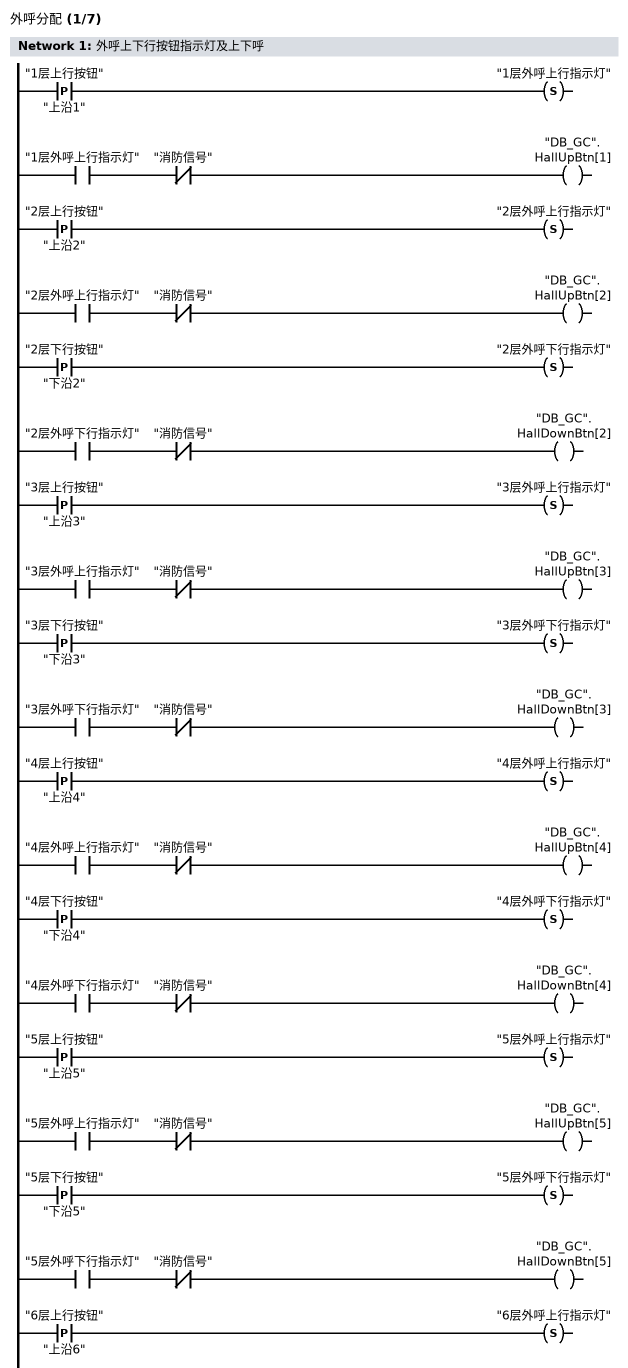
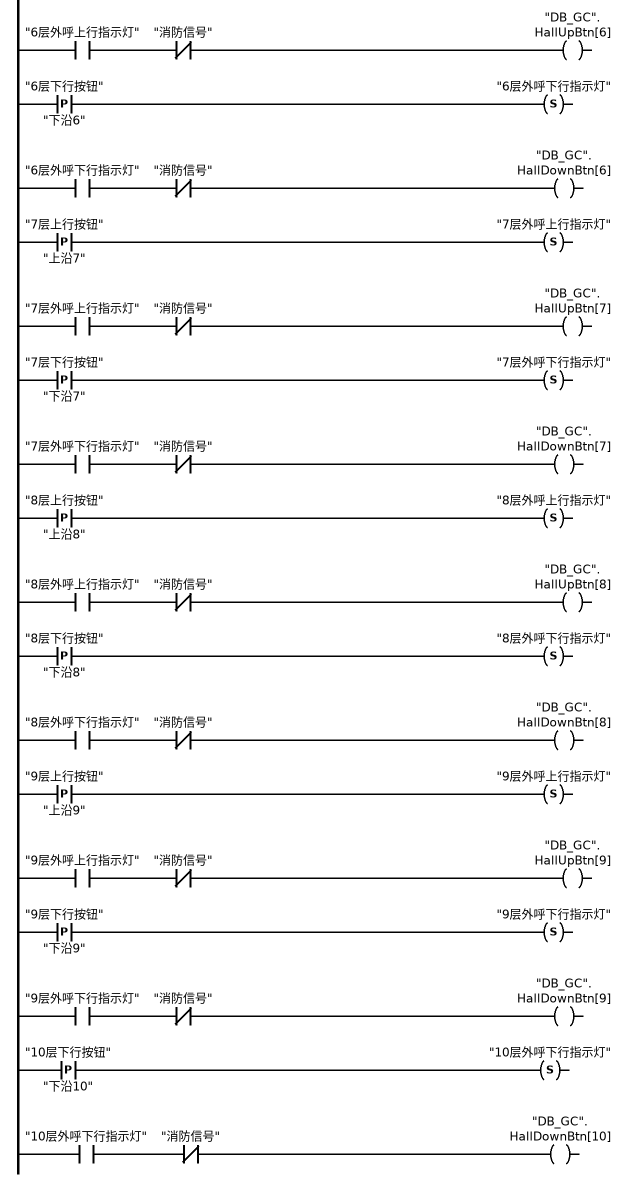
   RUNG wire#powerrail
      P_Contact(operand := "1层上行按钮", bit := "上沿1")
      S_Coil( "1层外呼上行指示灯" )
   END_RUNG
   RUNG wire#powerrail
      Contact( "1层外呼上行指示灯" )
      I_Contact( "消防信号" )
      Coil( "DB_GC".HallUpBtn[1] )
   END_RUNG
   RUNG wire#powerrail
      P_Contact(operand := "2层上行按钮", bit := "上沿2")
      S_Coil( "2层外呼上行指示灯" )
   END_RUNG
   RUNG wire#powerrail
      Contact( "2层外呼上行指示灯" )
      I_Contact( "消防信号" )
      Coil( "DB_GC".HallUpBtn[2] )
   END_RUNG
   RUNG wire#powerrail
      P_Contact(operand := "2层下行按钮", bit := "下沿2")
      S_Coil( "2层外呼下行指示灯" )
   END_RUNG
   RUNG wire#powerrail
      Contact( "2层外呼下行指示灯" )
      I_Contact( "消防信号" )
      Coil( "DB_GC".HallDownBtn[2] )
   END_RUNG
   RUNG wire#powerrail
      P_Contact(operand := "3层上行按钮", bit := "上沿3")
      S_Coil( "3层外呼上行指示灯" )
   END_RUNG
   RUNG wire#powerrail
      Contact( "3层外呼上行指示灯" )
      I_Contact( "消防信号" )
      Coil( "DB_GC".HallUpBtn[3] )
   END_RUNG
   RUNG wire#powerrail
      P_Contact(operand := "3层下行按钮", bit := "下沿3")
      S_Coil( "3层外呼下行指示灯" )
   END_RUNG
   RUNG wire#powerrail
      Contact( "3层外呼下行指示灯" )
      I_Contact( "消防信号" )
      Coil( "DB_GC".HallDownBtn[3] )
   END_RUNG
   RUNG wire#powerrail
      P_Contact(operand := "4层上行按钮", bit := "上沿4")
      S_Coil( "4层外呼上行指示灯" )
   END_RUNG
   RUNG wire#powerrail
      Contact( "4层外呼上行指示灯" )
      I_Contact( "消防信号" )
      Coil( "DB_GC".HallUpBtn[4] )
   END_RUNG
   RUNG wire#powerrail
      P_Contact(operand := "4层下行按钮", bit := "下沿4")
      S_Coil( "4层外呼下行指示灯" )
   END_RUNG
   RUNG wire#powerrail
      Contact( "4层外呼下行指示灯" )
      I_Contact( "消防信号" )
      Coil( "DB_GC".HallDownBtn[4] )
   END_RUNG
   RUNG wire#powerrail
      P_Contact(operand := "5层上行按钮", bit := "上沿5")
      S_Coil( "5层外呼上行指示灯" )
   END_RUNG
   RUNG wire#powerrail
      Contact( "5层外呼上行指示灯" )
      I_Contact( "消防信号" )
      Coil( "DB_GC".HallUpBtn[5] )
   END_RUNG
   RUNG wire#powerrail
      P_Contact(operand := "5层下行按钮", bit := "下沿5")
      S_Coil( "5层外呼下行指示灯" )
   END_RUNG
   RUNG wire#powerrail
      Contact( "5层外呼下行指示灯" )
      I_Contact( "消防信号" )
      Coil( "DB_GC".HallDownBtn[5] )
   END_RUNG
   RUNG wire#powerrail
      P_Contact(operand := "6层上行按钮", bit := "上沿6")
      S_Coil( "6层外呼上行指示灯" )
   END_RUNG
   RUNG wire#powerrail
      Contact( "6层外呼上行指示灯" )
      I_Contact( "消防信号" )
      Coil( "DB_GC".HallUpBtn[6] )
   END_RUNG
   RUNG wire#powerrail
      P_Contact(operand := "6层下行按钮", bit := "下沿6")
      S_Coil( "6层外呼下行指示灯" )
   END_RUNG
   RUNG wire#powerrail
      Contact( "6层外呼下行指示灯" )
      I_Contact( "消防信号" )
      Coil( "DB_GC".HallDownBtn[6] )
   END_RUNG
   RUNG wire#powerrail
      P_Contact(operand := "7层上行按钮", bit := "上沿7")
      S_Coil( "7层外呼上行指示灯" )
   END_RUNG
   RUNG wire#powerrail
      Contact( "7层外呼上行指示灯" )
      I_Contact( "消防信号" )
      Coil( "DB_GC".HallUpBtn[7] )
   END_RUNG
   RUNG wire#powerrail
      P_Contact(operand := "7层下行按钮", bit := "下沿7")
      S_Coil( "7层外呼下行指示灯" )
   END_RUNG
   RUNG wire#powerrail
      Contact( "7层外呼下行指示灯" )
      I_Contact( "消防信号" )
      Coil( "DB_GC".HallDownBtn[7] )
   END_RUNG
   RUNG wire#powerrail
      P_Contact(operand := "8层上行按钮", bit := "上沿8")
      S_Coil( "8层外呼上行指示灯" )
   END_RUNG
   RUNG wire#powerrail
      Contact( "8层外呼上行指示灯" )
      I_Contact( "消防信号" )
      Coil( "DB_GC".HallUpBtn[8] )
   END_RUNG
   RUNG wire#powerrail
      P_Contact(operand := "8层下行按钮", bit := "下沿8")
      S_Coil( "8层外呼下行指示灯" )
   END_RUNG
   RUNG wire#powerrail
      Contact( "8层外呼下行指示灯" )
      I_Contact( "消防信号" )
      Coil( "DB_GC".HallDownBtn[8] )
   END_RUNG
   RUNG wire#powerrail
      P_Contact(operand := "9层上行按钮", bit := "上沿9")
      S_Coil( "9层外呼上行指示灯" )
   END_RUNG
   RUNG wire#powerrail
      Contact( "9层外呼上行指示灯" )
      I_Contact( "消防信号" )
      Coil( "DB_GC".HallUpBtn[9] )
   END_RUNG
   RUNG wire#powerrail
      P_Contact(operand := "9层下行按钮", bit := "下沿9")
      S_Coil( "9层外呼下行指示灯" )
   END_RUNG
   RUNG wire#powerrail
      Contact( "9层外呼下行指示灯" )
      I_Contact( "消防信号" )
      Coil( "DB_GC".HallDownBtn[9] )
   END_RUNG
   RUNG wire#powerrail
      P_Contact(operand := "10层下行按钮", bit := "下沿10")
      S_Coil( "10层外呼下行指示灯" )
   END_RUNG
   RUNG wire#powerrail
      Contact( "10层外呼下行指示灯" )
      I_Contact( "消防信号" )
      Coil( "DB_GC".HallDownBtn[10] )
   END_RUNG
   // the same network as SCL:
   #_w1 := "1层上行按钮" AND NOT "上沿1";   // rising edge of "1层上行按钮"
   "上沿1" := "1层上行按钮";
   IF #_w1 THEN "1层外呼上行指示灯" := TRUE; END_IF;
   "DB_GC".HallUpBtn[1] := "1层外呼上行指示灯" AND NOT "消防信号";
   #_w2 := "2层上行按钮" AND NOT "上沿2";   // rising edge of "2层上行按钮"
   "上沿2" := "2层上行按钮";
   IF #_w2 THEN "2层外呼上行指示灯" := TRUE; END_IF;
   "DB_GC".HallUpBtn[2] := "2层外呼上行指示灯" AND NOT "消防信号";
   #_w3 := "2层下行按钮" AND NOT "下沿2";   // rising edge of "2层下行按钮"
   "下沿2" := "2层下行按钮";
   IF #_w3 THEN "2层外呼下行指示灯" := TRUE; END_IF;
   "DB_GC".HallDownBtn[2] := "2层外呼下行指示灯" AND NOT "消防信号";
   #_w4 := "3层上行按钮" AND NOT "上沿3";   // rising edge of "3层上行按钮"
   "上沿3" := "3层上行按钮";
   IF #_w4 THEN "3层外呼上行指示灯" := TRUE; END_IF;
   "DB_GC".HallUpBtn[3] := "3层外呼上行指示灯" AND NOT "消防信号";
   #_w5 := "3层下行按钮" AND NOT "下沿3";   // rising edge of "3层下行按钮"
   "下沿3" := "3层下行按钮";
   IF #_w5 THEN "3层外呼下行指示灯" := TRUE; END_IF;
   "DB_GC".HallDownBtn[3] := "3层外呼下行指示灯" AND NOT "消防信号";
   #_w6 := "4层上行按钮" AND NOT "上沿4";   // rising edge of "4层上行按钮"
   "上沿4" := "4层上行按钮";
   IF #_w6 THEN "4层外呼上行指示灯" := TRUE; END_IF;
   "DB_GC".HallUpBtn[4] := "4层外呼上行指示灯" AND NOT "消防信号";
   #_w7 := "4层下行按钮" AND NOT "下沿4";   // rising edge of "4层下行按钮"
   "下沿4" := "4层下行按钮";
   IF #_w7 THEN "4层外呼下行指示灯" := TRUE; END_IF;
   "DB_GC".HallDownBtn[4] := "4层外呼下行指示灯" AND NOT "消防信号";
   #_w8 := "5层上行按钮" AND NOT "上沿5";   // rising edge of "5层上行按钮"
   "上沿5" := "5层上行按钮";
   IF #_w8 THEN "5层外呼上行指示灯" := TRUE; END_IF;
   "DB_GC".HallUpBtn[5] := "5层外呼上行指示灯" AND NOT "消防信号";
   #_w9 := "5层下行按钮" AND NOT "下沿5";   // rising edge of "5层下行按钮"
   "下沿5" := "5层下行按钮";
   IF #_w9 THEN "5层外呼下行指示灯" := TRUE; END_IF;
   "DB_GC".HallDownBtn[5] := "5层外呼下行指示灯" AND NOT "消防信号";
   #_w10 := "6层上行按钮" AND NOT "上沿6";   // rising edge of "6层上行按钮"
   "上沿6" := "6层上行按钮";
   IF #_w10 THEN "6层外呼上行指示灯" := TRUE; END_IF;
   "DB_GC".HallUpBtn[6] := "6层外呼上行指示灯" AND NOT "消防信号";
   #_w11 := "6层下行按钮" AND NOT "下沿6";   // rising edge of "6层下行按钮"
   "下沿6" := "6层下行按钮";
   IF #_w11 THEN "6层外呼下行指示灯" := TRUE; END_IF;
   "DB_GC".HallDownBtn[6] := "6层外呼下行指示灯" AND NOT "消防信号";
   #_w12 := "7层上行按钮" AND NOT "上沿7";   // rising edge of "7层上行按钮"
   "上沿7" := "7层上行按钮";
   IF #_w12 THEN "7层外呼上行指示灯" := TRUE; END_IF;
   "DB_GC".HallUpBtn[7] := "7层外呼上行指示灯" AND NOT "消防信号";
   #_w13 := "7层下行按钮" AND NOT "下沿7";   // rising edge of "7层下行按钮"
   "下沿7" := "7层下行按钮";
   IF #_w13 THEN "7层外呼下行指示灯" := TRUE; END_IF;
   "DB_GC".HallDownBtn[7] := "7层外呼下行指示灯" AND NOT "消防信号";
   #_w14 := "8层上行按钮" AND NOT "上沿8";   // rising edge of "8层上行按钮"
   "上沿8" := "8层上行按钮";
   IF #_w14 THEN "8层外呼上行指示灯" := TRUE; END_IF;
   "DB_GC".HallUpBtn[8] := "8层外呼上行指示灯" AND NOT "消防信号";
   #_w15 := "8层下行按钮" AND NOT "下沿8";   // rising edge of "8层下行按钮"
   "下沿8" := "8层下行按钮";
   IF #_w15 THEN "8层外呼下行指示灯" := TRUE; END_IF;
   "DB_GC".HallDownBtn[8] := "8层外呼下行指示灯" AND NOT "消防信号";
   #_w16 := "9层上行按钮" AND NOT "上沿9";   // rising edge of "9层上行按钮"
   "上沿9" := "9层上行按钮";
   IF #_w16 THEN "9层外呼上行指示灯" := TRUE; END_IF;
   "DB_GC".HallUpBtn[9] := "9层外呼上行指示灯" AND NOT "消防信号";
   #_w17 := "9层下行按钮" AND NOT "下沿9";   // rising edge of "9层下行按钮"
   "下沿9" := "9层下行按钮";
   IF #_w17 THEN "9层外呼下行指示灯" := TRUE; END_IF;
   "DB_GC".HallDownBtn[9] := "9层外呼下行指示灯" AND NOT "消防信号";
   #_w18 := "10层下行按钮" AND NOT "下沿10";   // rising edge of "10层下行按钮"
   "下沿10" := "10层下行按钮";
   IF #_w18 THEN "10层外呼下行指示灯" := TRUE; END_IF;
   "DB_GC".HallDownBtn[10] := "10层外呼下行指示灯" AND NOT "消防信号";
END_REGION

REGION Network 2: 1号梯内呼指示灯绑定
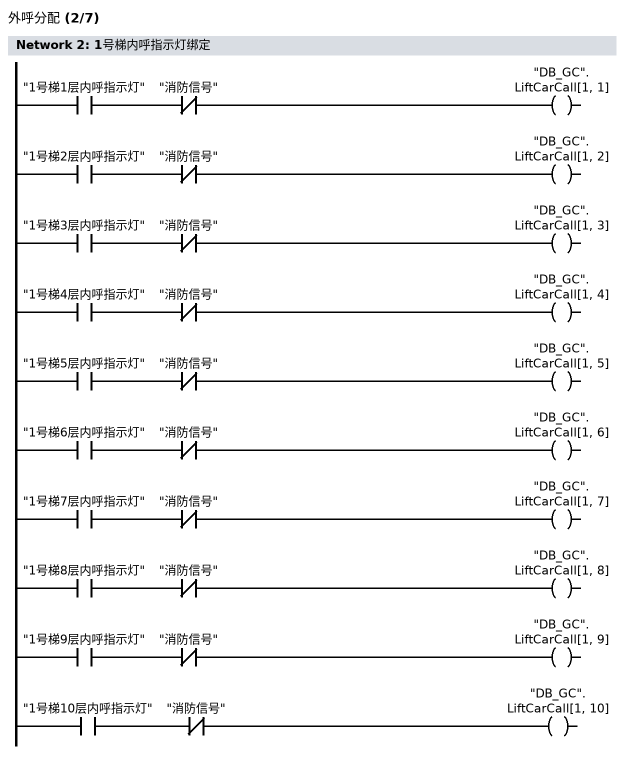
   RUNG wire#powerrail
      Contact( "1号梯1层内呼指示灯" )
      I_Contact( "消防信号" )
      Coil( "DB_GC".LiftCarCall[1, 1] )
   END_RUNG
   RUNG wire#powerrail
      Contact( "1号梯2层内呼指示灯" )
      I_Contact( "消防信号" )
      Coil( "DB_GC".LiftCarCall[1, 2] )
   END_RUNG
   RUNG wire#powerrail
      Contact( "1号梯3层内呼指示灯" )
      I_Contact( "消防信号" )
      Coil( "DB_GC".LiftCarCall[1, 3] )
   END_RUNG
   RUNG wire#powerrail
      Contact( "1号梯4层内呼指示灯" )
      I_Contact( "消防信号" )
      Coil( "DB_GC".LiftCarCall[1, 4] )
   END_RUNG
   RUNG wire#powerrail
      Contact( "1号梯5层内呼指示灯" )
      I_Contact( "消防信号" )
      Coil( "DB_GC".LiftCarCall[1, 5] )
   END_RUNG
   RUNG wire#powerrail
      Contact( "1号梯6层内呼指示灯" )
      I_Contact( "消防信号" )
      Coil( "DB_GC".LiftCarCall[1, 6] )
   END_RUNG
   RUNG wire#powerrail
      Contact( "1号梯7层内呼指示灯" )
      I_Contact( "消防信号" )
      Coil( "DB_GC".LiftCarCall[1, 7] )
   END_RUNG
   RUNG wire#powerrail
      Contact( "1号梯8层内呼指示灯" )
      I_Contact( "消防信号" )
      Coil( "DB_GC".LiftCarCall[1, 8] )
   END_RUNG
   RUNG wire#powerrail
      Contact( "1号梯9层内呼指示灯" )
      I_Contact( "消防信号" )
      Coil( "DB_GC".LiftCarCall[1, 9] )
   END_RUNG
   RUNG wire#powerrail
      Contact( "1号梯10层内呼指示灯" )
      I_Contact( "消防信号" )
      Coil( "DB_GC".LiftCarCall[1, 10] )
   END_RUNG
   // the same network as SCL:
   "DB_GC".LiftCarCall[1, 1] := "1号梯1层内呼指示灯" AND NOT "消防信号";
   "DB_GC".LiftCarCall[1, 2] := "1号梯2层内呼指示灯" AND NOT "消防信号";
   "DB_GC".LiftCarCall[1, 3] := "1号梯3层内呼指示灯" AND NOT "消防信号";
   "DB_GC".LiftCarCall[1, 4] := "1号梯4层内呼指示灯" AND NOT "消防信号";
   "DB_GC".LiftCarCall[1, 5] := "1号梯5层内呼指示灯" AND NOT "消防信号";
   "DB_GC".LiftCarCall[1, 6] := "1号梯6层内呼指示灯" AND NOT "消防信号";
   "DB_GC".LiftCarCall[1, 7] := "1号梯7层内呼指示灯" AND NOT "消防信号";
   "DB_GC".LiftCarCall[1, 8] := "1号梯8层内呼指示灯" AND NOT "消防信号";
   "DB_GC".LiftCarCall[1, 9] := "1号梯9层内呼指示灯" AND NOT "消防信号";
   "DB_GC".LiftCarCall[1, 10] := "1号梯10层内呼指示灯" AND NOT "消防信号";
END_REGION

REGION Network 3: 2号梯内呼指示灯绑定
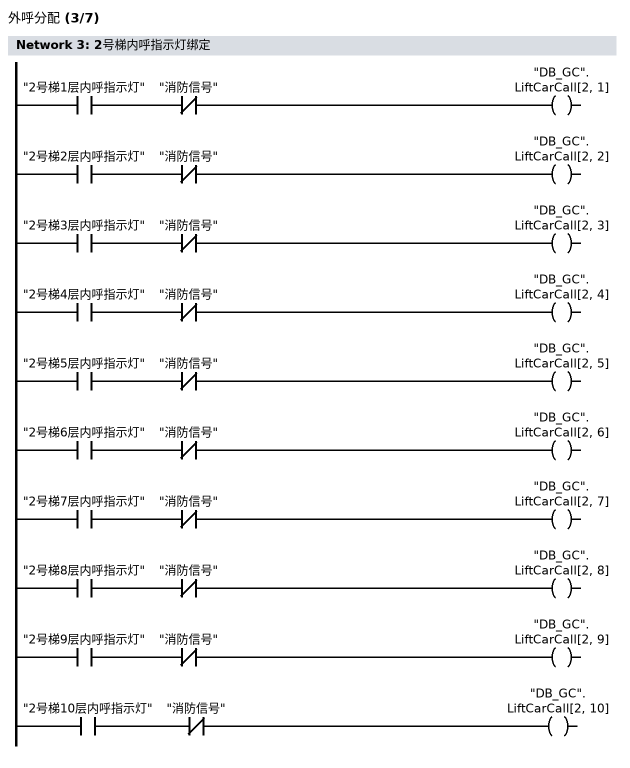
   RUNG wire#powerrail
      Contact( "2号梯1层内呼指示灯" )
      I_Contact( "消防信号" )
      Coil( "DB_GC".LiftCarCall[2, 1] )
   END_RUNG
   RUNG wire#powerrail
      Contact( "2号梯2层内呼指示灯" )
      I_Contact( "消防信号" )
      Coil( "DB_GC".LiftCarCall[2, 2] )
   END_RUNG
   RUNG wire#powerrail
      Contact( "2号梯3层内呼指示灯" )
      I_Contact( "消防信号" )
      Coil( "DB_GC".LiftCarCall[2, 3] )
   END_RUNG
   RUNG wire#powerrail
      Contact( "2号梯4层内呼指示灯" )
      I_Contact( "消防信号" )
      Coil( "DB_GC".LiftCarCall[2, 4] )
   END_RUNG
   RUNG wire#powerrail
      Contact( "2号梯5层内呼指示灯" )
      I_Contact( "消防信号" )
      Coil( "DB_GC".LiftCarCall[2, 5] )
   END_RUNG
   RUNG wire#powerrail
      Contact( "2号梯6层内呼指示灯" )
      I_Contact( "消防信号" )
      Coil( "DB_GC".LiftCarCall[2, 6] )
   END_RUNG
   RUNG wire#powerrail
      Contact( "2号梯7层内呼指示灯" )
      I_Contact( "消防信号" )
      Coil( "DB_GC".LiftCarCall[2, 7] )
   END_RUNG
   RUNG wire#powerrail
      Contact( "2号梯8层内呼指示灯" )
      I_Contact( "消防信号" )
      Coil( "DB_GC".LiftCarCall[2, 8] )
   END_RUNG
   RUNG wire#powerrail
      Contact( "2号梯9层内呼指示灯" )
      I_Contact( "消防信号" )
      Coil( "DB_GC".LiftCarCall[2, 9] )
   END_RUNG
   RUNG wire#powerrail
      Contact( "2号梯10层内呼指示灯" )
      I_Contact( "消防信号" )
      Coil( "DB_GC".LiftCarCall[2, 10] )
   END_RUNG
   // the same network as SCL:
   "DB_GC".LiftCarCall[2, 1] := "2号梯1层内呼指示灯" AND NOT "消防信号";
   "DB_GC".LiftCarCall[2, 2] := "2号梯2层内呼指示灯" AND NOT "消防信号";
   "DB_GC".LiftCarCall[2, 3] := "2号梯3层内呼指示灯" AND NOT "消防信号";
   "DB_GC".LiftCarCall[2, 4] := "2号梯4层内呼指示灯" AND NOT "消防信号";
   "DB_GC".LiftCarCall[2, 5] := "2号梯5层内呼指示灯" AND NOT "消防信号";
   "DB_GC".LiftCarCall[2, 6] := "2号梯6层内呼指示灯" AND NOT "消防信号";
   "DB_GC".LiftCarCall[2, 7] := "2号梯7层内呼指示灯" AND NOT "消防信号";
   "DB_GC".LiftCarCall[2, 8] := "2号梯8层内呼指示灯" AND NOT "消防信号";
   "DB_GC".LiftCarCall[2, 9] := "2号梯9层内呼指示灯" AND NOT "消防信号";
   "DB_GC".LiftCarCall[2, 10] := "2号梯10层内呼指示灯" AND NOT "消防信号";
END_REGION

